// TIA Portal V17 export
// export: Created 2023-12-22T15:05:25.6828662Z, ExportSetting WithDefaults, DisplayName Totally Integrated Automation Portal, DisplayVersion V17, DisplayName TIA Portal Openness, DisplayVersion V17, DisplayName TIA Portal Version Control Interface, DisplayVersion V17, DisplayName STEP 7 Professional, DisplayVersion V17, DisplayName STEP 7 Safety, DisplayVersion V17, DisplayName WinCC Advanced, DisplayVersion V17
FUNCTION_BLOCK "Block_Line"   // FB12, LAD
{ S7_Optimized_Access := 'TRUE' }
VERSION : 0.1
// stored: AutoNumber true, IsIECCheckEnabled false, IsRetainMemResEnabled false, MemoryReserve 100, SetENOAutomatically false, UDAEnableTagReadback false
   VAR_INPUT
      Flow : Real;   // Расходомер принимающей трубы
      SP_C : Real := 0.01;   // Уставка дозации, % масс, 0.05-1
      PE : Real;   // Датчик давления
      ALLS : Bool;   // Авариййный нижний уровень бака
      RT : Bool;   // Ротаметр
      RM : Bool;   // Датчик протока вместо расходомера
      KC_ON : Bool;   // Клапан открыт
      PE_LLS : Bool;
      PE_HHS : Bool;
   END_VAR
   VAR_OUTPUT
      KC_CMD : Bool;   // Открытие клапана
   END_VAR
   VAR_IN_OUT
      Report_H : "Line_Report";   // Разовый отчёт
   END_VAR
   VAR RETAIN
      LINE_NUMBER : Int;   // номер линии
   END_VAR
   VAR
      Start : Bool;   // Запуск линии
      Main_ON : Bool;   // Команда основного насоса
      Reserv_ON : Bool;   // Команда резервного насоса
   END_VAR
   VAR RETAIN
      Hand { S7_SetPoint := 'True'} : Bool;   // 1 - Задание скорости насосов в ручном режиме
      Choice_Tank : Bool;   // 0 - основной танк, 1 - резервный
      SP_Source { S7_SetPoint := 'True'} : Bool;   // 0 - по формуле расчета, 1 - равен входу Flow
      PID_Not_Use { S7_SetPoint := 'True'} : Bool;   // Использовать ПИД (0 - использовать, 1 - не использовать)
      Mode { S7_SetPoint := 'True'} : Bool;   // 0 - без разбаления, 1 - с разбавлением
      Mode_Local : Bool;   // Режим: 0 - местный, 1 - локальный
   END_VAR
   VAR
      Res_CMD : Bool;   // Команда ротации по наработке
      Res_ANY : Bool;   // Первый насос в резерве
      No_Water : Bool;   // Авария "Нет продукта" HMI
      Dry_Run : Bool;   // Авария "Нет протока, сухой ход" HMI
      Pump_Main_Alarm : Bool;   // Выходной сигнал аварии насоса 1
      Pump_Reserv_Alarm : Bool;   // Выходной сигнал аварии насоса 2
      Main_Line_Ok : Bool := true;   // Готовность основной линии
      Low_Stop : Bool;   // Остановка по низкому протоку
      RM_1_Alarm : Bool;   // Авария основного расходомера
      RM_2_Alarm : Bool;   // Авария дополнительного расходомера
   END_VAR
   VAR RETAIN
      RM_1_Report_DI { S7_SetPoint := 'True'} : Bool;   // Использовать импусльный сигнал для отчётов
      RM_2_Report_DI { S7_SetPoint := 'True'} : Bool;   // Использовать импусльный сигнал для отчётов
      RM_Weight { S7_SetPoint := 'True'} : Real := 1.0;   // Вес импульса
   END_VAR
   VAR
      Status_Main : Int;   // Статус основного насоса
      Status_Reserv : Int;   // Статус резервного насоса
      Events : Word;   // События линии
      SP_A : Real;   // Уставка авторежима
   END_VAR
   VAR RETAIN
      SP_M { S7_SetPoint := 'True'} : Real;   // Уставка ручного режима
      SP_min { S7_SetPoint := 'True'} : Real := 10.0;   // Минимальная скорость насоса
      SP_max { S7_SetPoint := 'True'} : Real := 1000.0;   // Максимальная скорость насоса
      PE_min { S7_SetPoint := 'True'} : Real := 0.15;   // Низкое давление в линии
      PE_max { S7_SetPoint := 'True'} : Real := 2.5;   // Высокое давление в линии
   END_VAR
   VAR
      Pump_SP : Real;   // Актуальная скорость насоса
   END_VAR
   VAR RETAIN
      D { S7_SetPoint := 'True'} : Real;   // Уставка дозы
      D_Num : Real;   // Количество замерок дозы
      D_Sum : Real;   // Общаяя сумма дозы
   END_VAR
   VAR
      C : Real;   // Рабочие данные о концентрации
   END_VAR
   VAR RETAIN
      C_Tank { S7_SetPoint := 'True'} : Real;   // Концентрация в резервном баке
   END_VAR
   VAR
      Flow_Line : Real;   // Расходомер, используемый в данный момент
      Flow_s { ExternalAccessible := 'False'; ExternalVisible := 'False'; ExternalWritable := 'False'} : Real;   // Переведенный в секунды
      Alarm_SP : Real;   // Аварийный коэфф соотношение уставки к реальной скорости насоса
   END_VAR
   VAR RETAIN
      Low_Flow { S7_SetPoint := 'True'} : Real;   // Низкий проток в основной линии
      Res_Main : Real;   // Наработка основного насоса
      Res_Reserv : Real;   // Наработка резревного насоса
      Res_SP { S7_SetPoint := 'True'} : Real;   // Уставка переключения по наработке
   END_VAR
   VAR
      Last_D : Real;   // Предъдущее значение дозы
      Last_SP : Real;   // Предъдущее значение расхода
   END_VAR
   VAR RETAIN
      Use : Struct   // Конфигурация
         RT { S7_SetPoint := 'True'} : Bool;   // Использование ротаметра
         RM { S7_SetPoint := 'True'} : Bool;   // Использование датчика протока вместо расходомера
         SP { S7_SetPoint := 'True'} : Bool := true;   // Использовать аналоговое регулирование
         Flow { S7_SetPoint := 'True'} : Bool := true;   // Использовать контрольный расходомер
         Res { S7_SetPoint := 'True'} : Bool;   // Использовать переключение по наработке
         DME { S7_SetPoint := 'True'} : Bool;   // Мембранные насосы
         PE { S7_SetPoint := 'True'} : Bool;
      END_STRUCT;
   END_VAR
   VAR
      Messages : Struct   // - Аварийные сообщения
         Low_Duct : Bool;   // Авария - низкий проток
         Low_Conc : Bool;   // Авария - низкая концентрация
         RT_ON : Bool;   // Авария - нет протока воды на ротаметре
         RT_OFF : Bool;   // Авария - поток воды не пропал на ротаметре
         RM_Error : Bool;   // Авария - неисправен расходомер
         PE_Low : Bool;   // Авария - низкое давление в линии
         PE_High : Bool;   // Авария - высокое давление в линии
         Alarm : Word;   // Слово аварий для панели
      END_STRUCT;
      Messages_Cancel : Struct   // - Отмена остановки
         Low_Duct : Bool;   // Авария - низкий проток
         Low_Conc : Bool;   // Авария - низкая концентрация
         RT_ON : Bool;   // Авария - нет протока воды на ротаметре
         RT_OFF : Bool;   // Авария - поток воды не пропал на ротаметре
         PE_Low : Bool;   // Авария - низкое давление в линии
         PE_High : Bool;   // Авария - высокое давление в линии
      END_STRUCT;
      Messages_Stop : Struct   // - Остановка по аварии
         Low_Duct : Bool;   // Авария - низкий проток
         Low_Conc : Bool;   // Авария - низкая концентрация
         RT_ON : Bool;   // Авария - нет протока воды на ротаметре
         RT_OFF : Bool;   // Авария - поток воды не пропал на ротаметре
         PE_Low : Bool;   // Авария - низкое давление в линии
         PE_High : Bool;   // Авария - высокое давление в линии
      END_STRUCT;
      Messages_Counter : Struct   // - Счётчик аварийных срабатываний
         Low_Duct : Int;   // Авария - низкий проток
         Low_Conc : Int;   // Авария - низкая концентрация
         RT_ON : Int;   // Авария - нет протока воды на ротаметре
         RT_OFF : Int;   // Авария - поток воды не пропал на ротаметре
         PE_Low : Int;   // Авария - низкое давление в линии
         PE_High : Int;   // Авария - высокое давление в линии
      END_STRUCT;
      Messages_Reset : Struct   // - Сброс счётчика
         Low_Duct : Bool;   // Авария - низкий проток
         Low_Conc : Bool;   // Авария - низкая концентрация
         RT_ON : Bool;   // Авария - нет протока воды на ротаметре
         RT_OFF : Bool;   // Авария - поток воды не пропал на ротаметре
         PE_Low : Bool;   // Авария - низкое давление в линии
         PE_High : Bool;   // Авария - высокое давление в линии
      END_STRUCT;
      Messages_REQ_Stop : Struct   // - Запрос остановки по аварии
         Low_Duct : Bool;   // Авария - низкий проток
         Low_Conc : Bool;   // Авария - низкая концентрация
         RT_ON : Bool;   // Авария - нет протока воды на ротаметре
         RT_OFF : Bool;   // Авария - поток воды не пропал на ротаметре
         PE_Low : Bool;   // Авария - низкое давление в линии
         PE_High : Bool;   // Авария - высокое давление в линии
      END_STRUCT;
      Timers_Stop : Array[0..5] of "Time_M";   // Таймеры останова
      Timers_Alm : Array[0..5] of "Time_M";   // Таймеры аварий
      T_Main_Alarm : "Time_M";   // Авария основного насоса по датчику протока
      T_Reserv_Alarm : "Time_M";   // Авария резервного насоса по датчику протока
      T_Main_Line_Ok : "Time_M";   // Таймер готовности основной линии
      T_No_Water : "Time_M";   // Нет продукта в баке
      T_Dry_Run : "Time_M";   // Нет протока в линии
      pos : Array[0..15] of Bool;   // Вспомогательные переменные
      PID { S7_SetPoint := 'True'} : "PID_ex";
      FlowMeter_1 { S7_SetPoint := 'True'} : "DRV_Flow_old";   // Расход 1
      FlowMeter_2 { S7_SetPoint := 'True'} : "DRV_Flow_old";   // Расход 2
   END_VAR
   VAR_TEMP
      ev : Bool;
      x : Real;
   END_VAR
   VAR CONSTANT
      "1s" : Real := 0.00028;
      "1m" : Real := 0.017;
   END_VAR
   // // Report_H.Res_1 : Резерв 1
   // // Report_H.Res_2 : Резерв 2
   VAR_TEMP   // added for the SCL form of the ladder/FBD networks
      _w1 : Bool;
      _w2 : Bool;
      _w3 : Bool;
      _w4 : Bool;
      _w5 : Bool;
      _w6 : Bool;
      _w7 : Bool;
      _w8 : Bool;
      _w9 : Bool;
      _w10 : Bool;
      _w11 : Bool;
      _w12 : Bool;
      _w13 : Bool;
      _w14 : Bool;
   END_VAR
BEGIN

REGION Network 1: Режим: 0 - местный, 1 - локальный
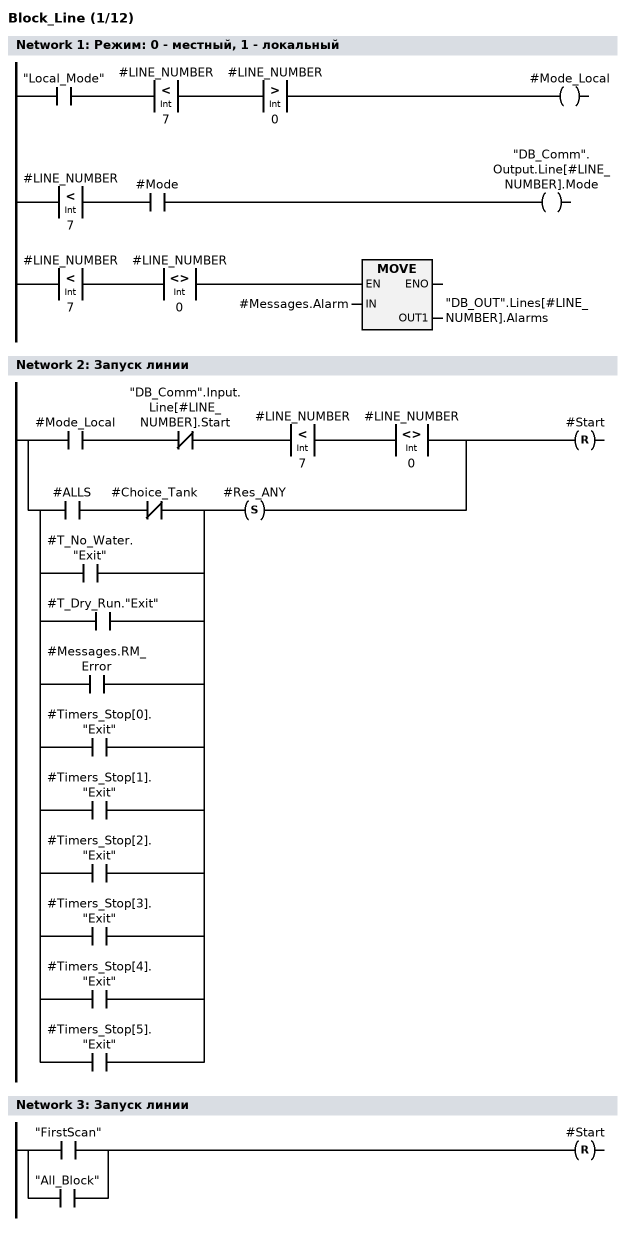
   RUNG wire#powerrail
      Contact( "Local_Mode" )
      { S7_Templates := "SrcType := Int" } LT_Contact(in1 := #LINE_NUMBER, in2 := 7)
      { S7_Templates := "SrcType := Int" } GT_Contact(in1 := #LINE_NUMBER, in2 := 0)
      Coil( #Mode_Local )
   END_RUNG
   RUNG wire#powerrail
      { S7_Templates := "SrcType := Int" } LT_Contact(in1 := #LINE_NUMBER, in2 := 7)
      Contact( #Mode )
      Coil( "DB_Comm".Output.Line[#LINE_NUMBER].Mode )
   END_RUNG
   RUNG wire#powerrail
      { S7_Templates := "SrcType := Int" } LT_Contact(in1 := #LINE_NUMBER, in2 := 7)
      { S7_Templates := "SrcType := Int" } NE_Contact(in1 := #LINE_NUMBER, in2 := 0)
      Move(in := #Messages.Alarm, out1 => "DB_OUT".Lines[#LINE_NUMBER].Alarms)
   END_RUNG
   // the same network as SCL:
   #Mode_Local := "Local_Mode" AND (#LINE_NUMBER < 7) AND (#LINE_NUMBER > 0);
   "DB_Comm".Output.Line[#LINE_NUMBER].Mode := (#LINE_NUMBER < 7) AND #Mode;
   IF (#LINE_NUMBER < 7) AND (#LINE_NUMBER <> 0) THEN
       "DB_OUT".Lines[#LINE_NUMBER].Alarms := #Messages.Alarm;
   END_IF;
END_REGION

REGION Network 2: Запуск линии
   RUNG wire#powerrail
      Contact( #Mode_Local )
      I_Contact( "DB_Comm".Input.Line[#LINE_NUMBER].Start )
      { S7_Templates := "SrcType := Int" } LT_Contact(in1 := #LINE_NUMBER, in2 := 7)
      { S7_Templates := "SrcType := Int" } NE_Contact(in1 := #LINE_NUMBER, in2 := 0)
      wire#w1
      R_Coil( #Start )
   END_RUNG
   RUNG wire#powerrail
      Contact( #ALLS )
      I_Contact( #Choice_Tank )
      wire#w2
      S_Coil( #Res_ANY )
   END_RUNG wire#w1
   RUNG wire#powerrail
      Contact( #T_No_Water."Exit" )
   END_RUNG wire#w2
   RUNG wire#powerrail
      Contact( #T_Dry_Run."Exit" )
   END_RUNG wire#w2
   RUNG wire#powerrail
      Contact( #Messages.RM_Error )
   END_RUNG wire#w2
   RUNG wire#powerrail
      Contact( #Timers_Stop[0]."Exit" )
   END_RUNG wire#w2
   RUNG wire#powerrail
      Contact( #Timers_Stop[1]."Exit" )
   END_RUNG wire#w2
   RUNG wire#powerrail
      Contact( #Timers_Stop[2]."Exit" )
   END_RUNG wire#w2
   RUNG wire#powerrail
      Contact( #Timers_Stop[3]."Exit" )
   END_RUNG wire#w2
   RUNG wire#powerrail
      Contact( #Timers_Stop[4]."Exit" )
   END_RUNG wire#w2
   RUNG wire#powerrail
      Contact( #Timers_Stop[5]."Exit" )
   END_RUNG wire#w2
   // the same network as SCL:
   #_w1 := (#ALLS AND NOT #Choice_Tank) OR #T_No_Water."Exit" OR #T_Dry_Run."Exit" OR #Messages.RM_Error OR #Timers_Stop[0]."Exit" OR #Timers_Stop[1]."Exit" OR #Timers_Stop[2]."Exit" OR #Timers_Stop[3]."Exit" OR #Timers_Stop[4]."Exit" OR #Timers_Stop[5]."Exit";
   IF #_w1 THEN #Res_ANY := TRUE; END_IF;
   IF (#Mode_Local AND NOT "DB_Comm".Input.Line[#LINE_NUMBER].Start AND (#LINE_NUMBER < 7) AND (#LINE_NUMBER <> 0)) OR #_w1 THEN
       #Start := FALSE;
   END_IF;
END_REGION

REGION Network 3: Запуск линии
   RUNG wire#powerrail
      Contact( "FirstScan" )
      wire#w1
      R_Coil( #Start )
   END_RUNG
   RUNG wire#powerrail
      Contact( "All_Block" )
   END_RUNG wire#w1
   // the same network as SCL:
   IF "FirstScan" OR "All_Block" THEN #Start := FALSE; END_IF;
END_REGION

REGION Network 4: Формирование событий линии
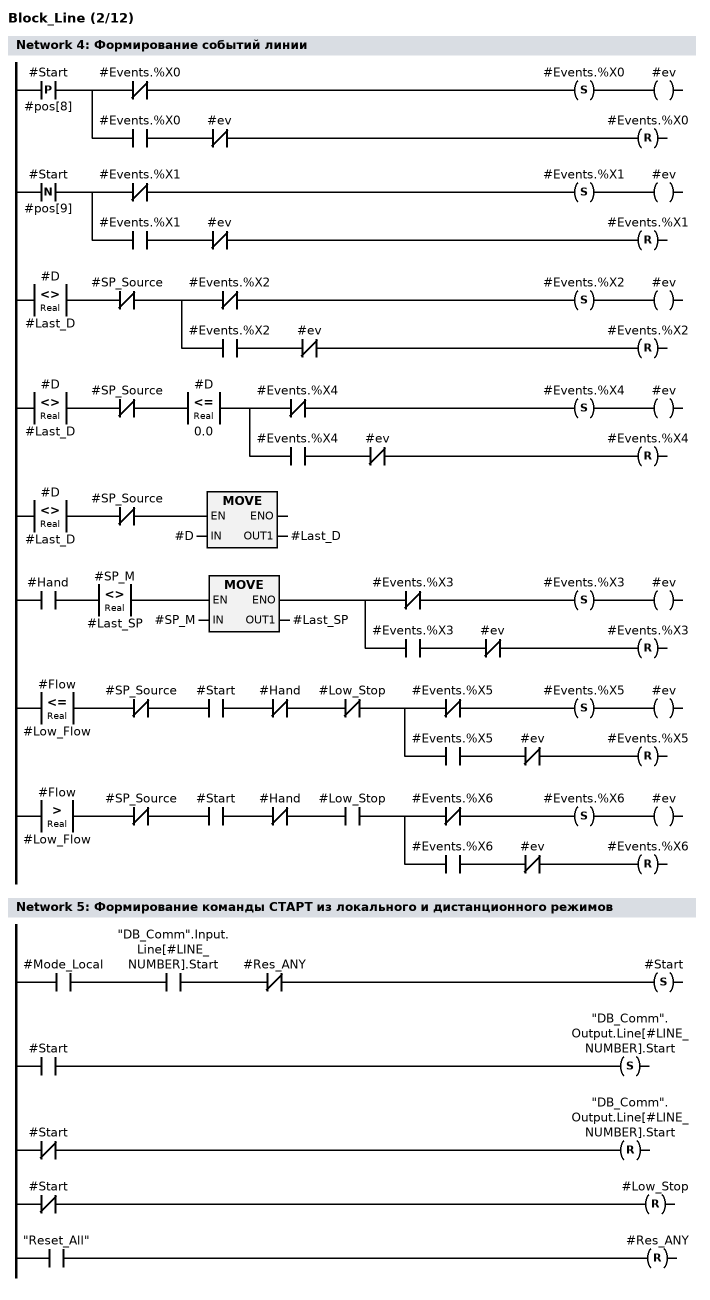
   RUNG wire#powerrail
      P_Contact(operand := #Start, bit := #pos[8])
      wire#w1
      I_Contact( #Events.%X0 )
      S_Coil( #Events.%X0 )
      Coil( #ev )
   END_RUNG
   RUNG wire#w1
      Contact( #Events.%X0 )
      I_Contact( #ev )
      R_Coil( #Events.%X0 )
   END_RUNG
   RUNG wire#powerrail
      N_Contact(operand := #Start, bit := #pos[9])
      wire#w2
      I_Contact( #Events.%X1 )
      S_Coil( #Events.%X1 )
      Coil( #ev )
   END_RUNG
   RUNG wire#w2
      Contact( #Events.%X1 )
      I_Contact( #ev )
      R_Coil( #Events.%X1 )
   END_RUNG
   RUNG wire#powerrail
      { S7_Templates := "SrcType := Real" } NE_Contact(in1 := #D, in2 := #Last_D)
      I_Contact( #SP_Source )
      wire#w3
      I_Contact( #Events.%X2 )
      S_Coil( #Events.%X2 )
      Coil( #ev )
   END_RUNG
   RUNG wire#w3
      Contact( #Events.%X2 )
      I_Contact( #ev )
      R_Coil( #Events.%X2 )
   END_RUNG
   RUNG wire#powerrail
      { S7_Templates := "SrcType := Real" } NE_Contact(in1 := #D, in2 := #Last_D)
      I_Contact( #SP_Source )
      { S7_Templates := "SrcType := Real" } LE_Contact(in1 := #D, in2 := 0.0)
      wire#w4
      I_Contact( #Events.%X4 )
      S_Coil( #Events.%X4 )
      Coil( #ev )
   END_RUNG
   RUNG wire#w4
      Contact( #Events.%X4 )
      I_Contact( #ev )
      R_Coil( #Events.%X4 )
   END_RUNG
   RUNG wire#powerrail
      { S7_Templates := "SrcType := Real" } NE_Contact(in1 := #D, in2 := #Last_D)
      I_Contact( #SP_Source )
      Move(in := #D, out1 => #Last_D)
   END_RUNG
   RUNG wire#powerrail
      Contact( #Hand )
      { S7_Templates := "SrcType := Real" } NE_Contact(in1 := #SP_M, in2 := #Last_SP)
      Move(in := #SP_M, out1 => #Last_SP)
      wire#w5
      I_Contact( #Events.%X3 )
      S_Coil( #Events.%X3 )
      Coil( #ev )
   END_RUNG
   RUNG wire#w5
      Contact( #Events.%X3 )
      I_Contact( #ev )
      R_Coil( #Events.%X3 )
   END_RUNG
   RUNG wire#powerrail
      { S7_Templates := "SrcType := Real" } LE_Contact(in1 := #Flow, in2 := #Low_Flow)
      I_Contact( #SP_Source )
      Contact( #Start )
      I_Contact( #Hand )
      I_Contact( #Low_Stop )
      wire#w6
      I_Contact( #Events.%X5 )
      S_Coil( #Events.%X5 )
      Coil( #ev )
   END_RUNG
   RUNG wire#w6
      Contact( #Events.%X5 )
      I_Contact( #ev )
      R_Coil( #Events.%X5 )
   END_RUNG
   RUNG wire#powerrail
      { S7_Templates := "SrcType := Real" } GT_Contact(in1 := #Flow, in2 := #Low_Flow)
      I_Contact( #SP_Source )
      Contact( #Start )
      I_Contact( #Hand )
      Contact( #Low_Stop )
      wire#w7
      I_Contact( #Events.%X6 )
      S_Coil( #Events.%X6 )
      Coil( #ev )
   END_RUNG
   RUNG wire#w7
      Contact( #Events.%X6 )
      I_Contact( #ev )
      R_Coil( #Events.%X6 )
   END_RUNG
   // the same network as SCL:
   #_w1 := #Start AND NOT #pos[8];   // rising edge of #Start
   #pos[8] := #Start;
   #_w2 := #_w1 AND NOT #Events.%X0;
   IF #_w2 THEN #Events.%X0 := TRUE; END_IF;
   #ev := #_w2;
   IF #_w1 AND #Events.%X0 AND NOT #ev THEN #Events.%X0 := FALSE; END_IF;
   #_w3 := NOT #Start AND #pos[9];   // falling edge of #Start
   #pos[9] := #Start;
   #_w4 := #_w3 AND NOT #Events.%X1;
   IF #_w4 THEN #Events.%X1 := TRUE; END_IF;
   #ev := #_w4;
   IF #_w3 AND #Events.%X1 AND NOT #ev THEN #Events.%X1 := FALSE; END_IF;
   #_w5 := (#D <> #Last_D) AND NOT #SP_Source;
   #_w6 := #_w5 AND NOT #Events.%X2;
   IF #_w6 THEN #Events.%X2 := TRUE; END_IF;
   #ev := #_w6;
   IF #_w5 AND #Events.%X2 AND NOT #ev THEN #Events.%X2 := FALSE; END_IF;
   #_w7 := (#D <> #Last_D) AND NOT #SP_Source AND (#D <= 0.0);
   #_w8 := #_w7 AND NOT #Events.%X4;
   IF #_w8 THEN #Events.%X4 := TRUE; END_IF;
   #ev := #_w8;
   IF #_w7 AND #Events.%X4 AND NOT #ev THEN #Events.%X4 := FALSE; END_IF;
   IF (#D <> #Last_D) AND NOT #SP_Source THEN #Last_D := #D; END_IF;
   #_w9 := #Hand AND (#SP_M <> #Last_SP);
   IF #_w9 THEN #Last_SP := #SP_M; END_IF;
   #_w10 := #_w9 AND NOT #Events.%X3;
   IF #_w10 THEN #Events.%X3 := TRUE; END_IF;
   #ev := #_w10;
   IF #_w9 AND #Events.%X3 AND NOT #ev THEN #Events.%X3 := FALSE; END_IF;
   #_w11 := (#Flow <= #Low_Flow) AND NOT #SP_Source AND #Start AND NOT #Hand AND NOT #Low_Stop;
   #_w12 := #_w11 AND NOT #Events.%X5;
   IF #_w12 THEN #Events.%X5 := TRUE; END_IF;
   #ev := #_w12;
   IF #_w11 AND #Events.%X5 AND NOT #ev THEN #Events.%X5 := FALSE; END_IF;
   #_w13 := (#Flow > #Low_Flow) AND NOT #SP_Source AND #Start AND NOT #Hand AND #Low_Stop;
   #_w14 := #_w13 AND NOT #Events.%X6;
   IF #_w14 THEN #Events.%X6 := TRUE; END_IF;
   #ev := #_w14;
   IF #_w13 AND #Events.%X6 AND NOT #ev THEN #Events.%X6 := FALSE; END_IF;
END_REGION

REGION Network 5: Формирование команды СТАРТ из локального и дистанционного режимов
   RUNG wire#powerrail
      Contact( #Mode_Local )
      Contact( "DB_Comm".Input.Line[#LINE_NUMBER].Start )
      I_Contact( #Res_ANY )
      S_Coil( #Start )
   END_RUNG
   RUNG wire#powerrail
      Contact( #Start )
      S_Coil( "DB_Comm".Output.Line[#LINE_NUMBER].Start )
   END_RUNG
   RUNG wire#powerrail
      I_Contact( #Start )
      R_Coil( "DB_Comm".Output.Line[#LINE_NUMBER].Start )
   END_RUNG
   RUNG wire#powerrail
      I_Contact( #Start )
      R_Coil( #Low_Stop )
   END_RUNG
   RUNG wire#powerrail
      Contact( "Reset_All" )
      R_Coil( #Res_ANY )
   END_RUNG
   // the same network as SCL:
   IF #Mode_Local AND "DB_Comm".Input.Line[#LINE_NUMBER].Start AND NOT #Res_ANY THEN #Start := TRUE; END_IF;
   IF #Start THEN "DB_Comm".Output.Line[#LINE_NUMBER].Start := TRUE; END_IF;
   IF NOT #Start THEN
       "DB_Comm".Output.Line[#LINE_NUMBER].Start := FALSE;
       #Low_Stop := FALSE;
   END_IF;
   IF "Reset_All" THEN #Res_ANY := FALSE; END_IF;
END_REGION

REGION Network 6: Старт - выбора насоса
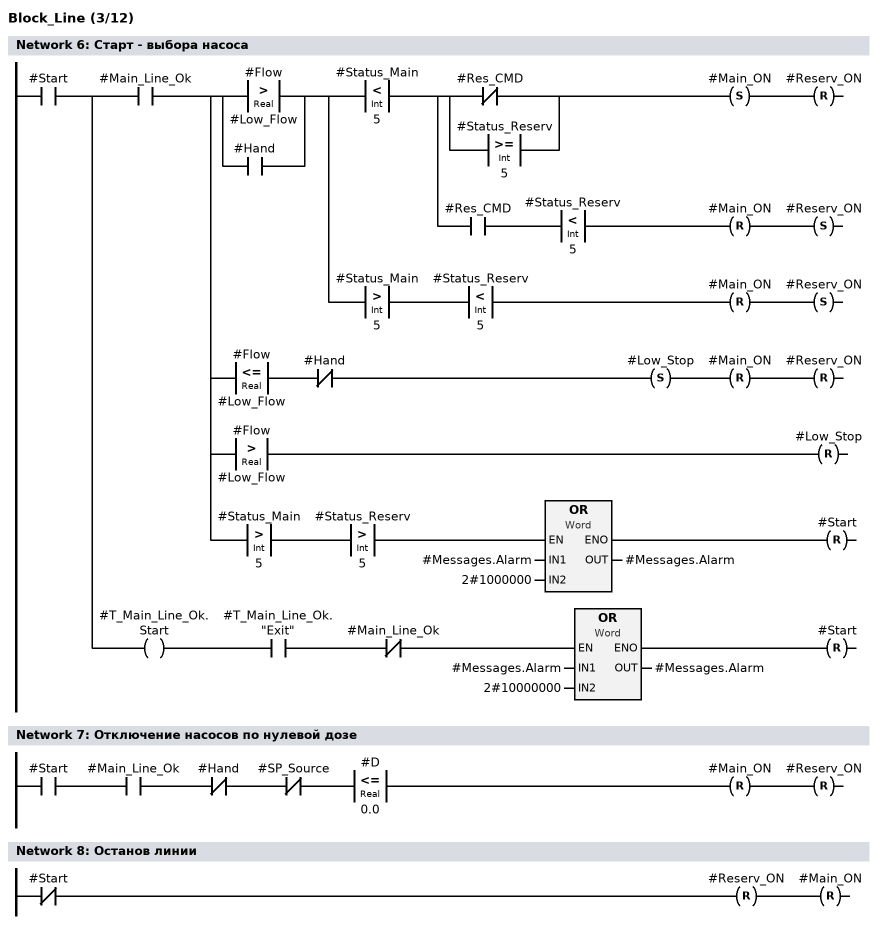
   #_w1 := #Start AND #Main_Line_Ok;
   #_w2 := #_w1 AND ((#Flow > #Low_Flow) OR #Hand);
   #_w3 := #_w2 AND (#Status_Main < 5);
   IF #_w3 AND (NOT #Res_CMD OR (#Status_Reserv >= 5)) THEN
       #Main_ON := TRUE;
       #Reserv_ON := FALSE;
   END_IF;
   IF #_w3 AND #Res_CMD AND (#Status_Reserv < 5) THEN
       #Main_ON := FALSE;
       #Reserv_ON := TRUE;
   END_IF;
   IF #_w2 AND (#Status_Main > 5) AND (#Status_Reserv < 5) THEN
       #Main_ON := FALSE;
       #Reserv_ON := TRUE;
   END_IF;
   IF #_w1 AND (#Flow <= #Low_Flow) AND NOT #Hand THEN
       #Low_Stop := TRUE;
       #Main_ON := FALSE;
       #Reserv_ON := FALSE;
   END_IF;
   IF #_w1 AND (#Flow > #Low_Flow) THEN #Low_Stop := FALSE; END_IF;
   IF #_w1 AND (#Status_Main > 5) AND (#Status_Reserv > 5) THEN
       #Messages.Alarm := #Messages.Alarm OR 2#1000000;
   END_IF;
   #_w4 := #Start;
   IF #_w1 AND (#Status_Main > 5) AND (#Status_Reserv > 5) THEN #Start := FALSE; END_IF;
   #T_Main_Line_Ok.Start := #_w4;
   IF #_w4 AND #T_Main_Line_Ok."Exit" AND NOT #Main_Line_Ok THEN
       #Messages.Alarm := #Messages.Alarm OR 2#10000000;
       #Start := FALSE;
   END_IF;
END_REGION

REGION Network 7: Отключение насосов по нулевой дозе
   RUNG wire#powerrail
      Contact( #Start )
      Contact( #Main_Line_Ok )
      I_Contact( #Hand )
      I_Contact( #SP_Source )
      { S7_Templates := "SrcType := Real" } LE_Contact(in1 := #D, in2 := 0.0)
      R_Coil( #Main_ON )
      R_Coil( #Reserv_ON )
   END_RUNG
   // the same network as SCL:
   IF #Start AND #Main_Line_Ok AND NOT #Hand AND NOT #SP_Source AND (#D <= 0.0) THEN
       #Main_ON := FALSE;
       #Reserv_ON := FALSE;
   END_IF;
END_REGION

REGION Network 8: Останов линии
   RUNG wire#powerrail
      I_Contact( #Start )
      R_Coil( #Reserv_ON )
      R_Coil( #Main_ON )
   END_RUNG
   // the same network as SCL:
   IF NOT #Start THEN
       #Reserv_ON := FALSE;
       #Main_ON := FALSE;
   END_IF;
END_REGION

REGION Network 9: Подсчёт наработки насосов и управление выбором основного и резервного
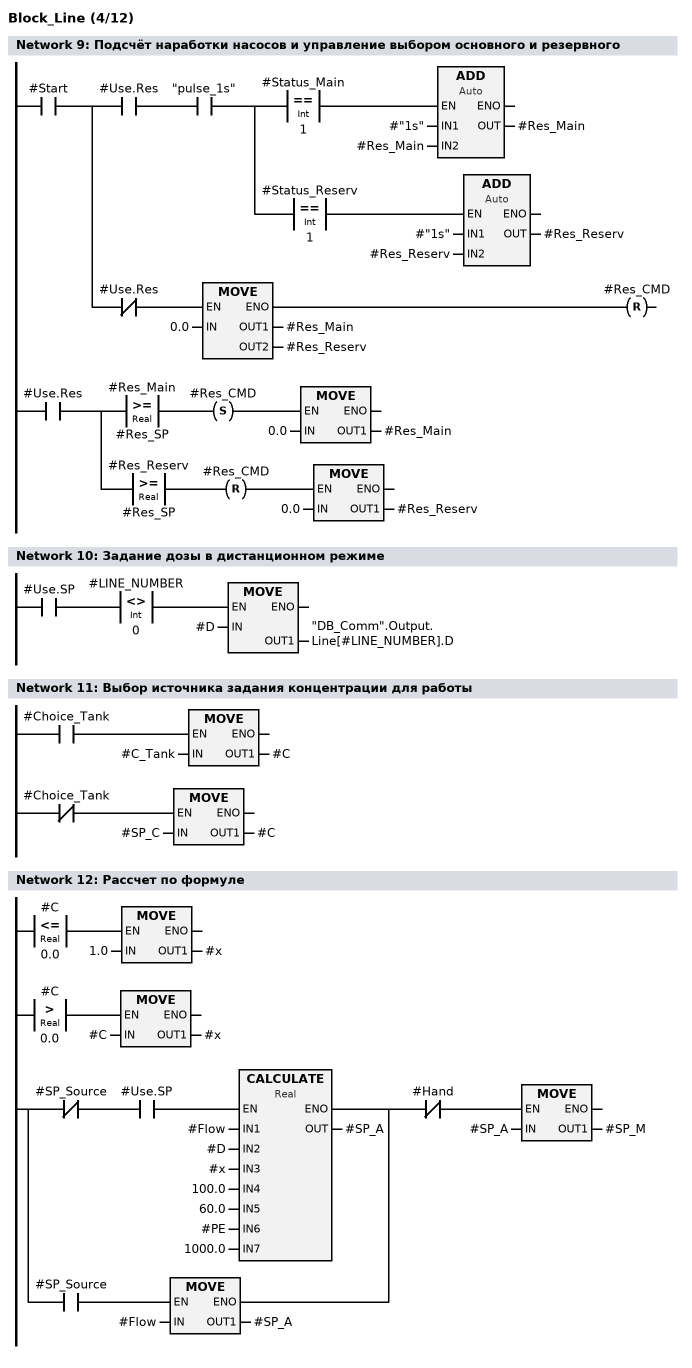
   RUNG wire#powerrail
      Contact( #Start )
      wire#w1
      Contact( #Use.Res )
      Contact( "pulse_1s" )
      wire#w2
      { S7_Templates := "SrcType := Int" } EQ_Contact(in1 := #Status_Main, in2 := 1)
      Add(in1 := #"1s", in2 := #Res_Main, out => #Res_Main)
   END_RUNG
   RUNG wire#w2
      { S7_Templates := "SrcType := Int" } EQ_Contact(in1 := #Status_Reserv, in2 := 1)
      Add(in1 := #"1s", in2 := #Res_Reserv, out => #Res_Reserv)
   END_RUNG
   RUNG wire#w1
      I_Contact( #Use.Res )
      Move(in := 0.0, out1 => #Res_Main, out2 => #Res_Reserv)
      R_Coil( #Res_CMD )
   END_RUNG
   RUNG wire#powerrail
      Contact( #Use.Res )
      wire#w3
      { S7_Templates := "SrcType := Real" } GE_Contact(in1 := #Res_Main, in2 := #Res_SP)
      S_Coil( #Res_CMD )
      Move(in := 0.0, out1 => #Res_Main)
   END_RUNG
   RUNG wire#w3
      { S7_Templates := "SrcType := Real" } GE_Contact(in1 := #Res_Reserv, in2 := #Res_SP)
      R_Coil( #Res_CMD )
      Move(in := 0.0, out1 => #Res_Reserv)
   END_RUNG
   // the same network as SCL:
   #_w1 := #Start AND #Use.Res AND "pulse_1s";
   IF #_w1 AND (#Status_Main = 1) THEN #Res_Main := #"1s" + #Res_Main; END_IF;
   IF #_w1 AND (#Status_Reserv = 1) THEN #Res_Reserv := #"1s" + #Res_Reserv; END_IF;
   IF #Start AND NOT #Use.Res THEN
       #Res_Main := 0.0;
       #Res_Reserv := 0.0;
       #Res_CMD := FALSE;
   END_IF;
   IF #Use.Res AND (#Res_Main >= #Res_SP) THEN
       #Res_CMD := TRUE;
       #Res_Main := 0.0;
   END_IF;
   IF #Use.Res AND (#Res_Reserv >= #Res_SP) THEN
       #Res_CMD := FALSE;
       #Res_Reserv := 0.0;
   END_IF;
END_REGION

REGION Network 10: Задание дозы в дистанционном режиме
   RUNG wire#powerrail
      Contact( #Use.SP )
      { S7_Templates := "SrcType := Int" } NE_Contact(in1 := #LINE_NUMBER, in2 := 0)
      Move(in := #D, out1 => "DB_Comm".Output.Line[#LINE_NUMBER].D)
   END_RUNG
   // the same network as SCL:
   IF #Use.SP AND (#LINE_NUMBER <> 0) THEN "DB_Comm".Output.Line[#LINE_NUMBER].D := #D; END_IF;
END_REGION

REGION Network 11: Выбор источника задания концентрации для работы
   RUNG wire#powerrail
      Contact( #Choice_Tank )
      Move(in := #C_Tank, out1 => #C)
   END_RUNG
   RUNG wire#powerrail
      I_Contact( #Choice_Tank )
      Move(in := #SP_C, out1 => #C)
   END_RUNG
   // the same network as SCL:
   IF #Choice_Tank THEN #C := #C_Tank; END_IF;
   IF NOT #Choice_Tank THEN #C := #SP_C; END_IF;
END_REGION

REGION Network 12: Рассчет по формуле
   RUNG wire#powerrail
      { S7_Templates := "SrcType := Real" } LE_Contact(in1 := #C, in2 := 0.0)
      Move(in := 1.0, out1 => #x)
   END_RUNG
   RUNG wire#powerrail
      { S7_Templates := "SrcType := Real" } GT_Contact(in1 := #C, in2 := 0.0)
      Move(in := #C, out1 => #x)
   END_RUNG
   RUNG wire#powerrail
      I_Contact( #SP_Source )
      Contact( #Use.SP )
      { S7_Templates := "SrcType := Real"; S7_Expression := "(IN2 * IN1) / ( IN3 / IN4) / (IN6 * IN7) / IN5" } Calculate(in1 := #Flow, in2 := #D, in3 := #x, in4 := 100.0, in5 := 60.0, in6 := #PE, in7 := 1000.0, out => #SP_A)
      wire#w1
      I_Contact( #Hand )
      Move(in := #SP_A, out1 => #SP_M)
   END_RUNG
   RUNG wire#powerrail
      Contact( #SP_Source )
      Move(in := #Flow, out1 => #SP_A)
   END_RUNG wire#w1
   // the same network as SCL:
   IF #C <= 0.0 THEN #x := 1.0; END_IF;
   IF #C > 0.0 THEN #x := #C; END_IF;
   #_w1 := NOT #SP_Source AND #Use.SP;
   IF #_w1 THEN #SP_A := (#D * #Flow) / ( #x / 100.0) / (#PE * 1000.0) / 60.0; END_IF;
   IF #SP_Source THEN #SP_A := #Flow; END_IF;
   IF (#_w1 OR #SP_Source) AND NOT #Hand THEN #SP_M := #SP_A; END_IF;
END_REGION

REGION Network 13: Выбор режима с разбавлением или без разбавления в дистанционном режиме
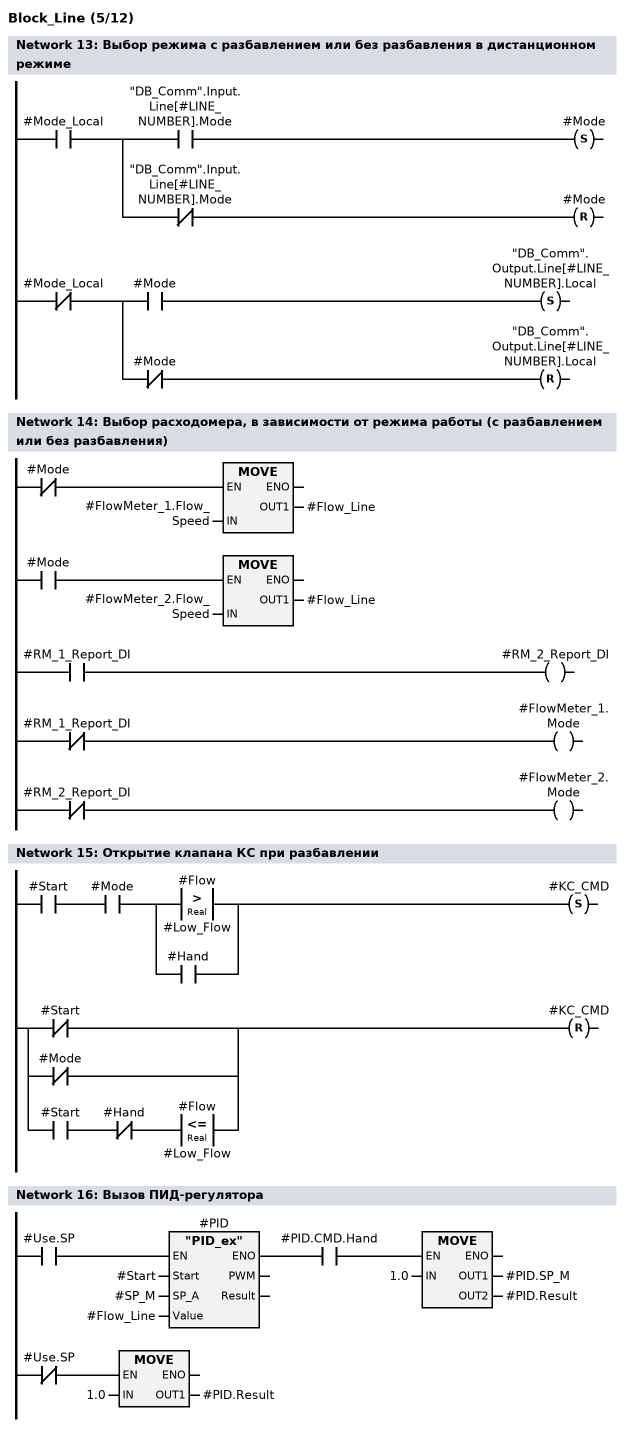
   RUNG wire#powerrail
      Contact( #Mode_Local )
      wire#w1
      Contact( "DB_Comm".Input.Line[#LINE_NUMBER].Mode )
      S_Coil( #Mode )
   END_RUNG
   RUNG wire#w1
      I_Contact( "DB_Comm".Input.Line[#LINE_NUMBER].Mode )
      R_Coil( #Mode )
   END_RUNG
   RUNG wire#powerrail
      I_Contact( #Mode_Local )
      wire#w2
      Contact( #Mode )
      S_Coil( "DB_Comm".Output.Line[#LINE_NUMBER].Local )
   END_RUNG
   RUNG wire#w2
      I_Contact( #Mode )
      R_Coil( "DB_Comm".Output.Line[#LINE_NUMBER].Local )
   END_RUNG
   // the same network as SCL:
   IF #Mode_Local AND "DB_Comm".Input.Line[#LINE_NUMBER].Mode THEN #Mode := TRUE; END_IF;
   IF #Mode_Local AND NOT "DB_Comm".Input.Line[#LINE_NUMBER].Mode THEN #Mode := FALSE; END_IF;
   IF NOT #Mode_Local AND #Mode THEN "DB_Comm".Output.Line[#LINE_NUMBER].Local := TRUE; END_IF;
   IF NOT #Mode_Local AND NOT #Mode THEN "DB_Comm".Output.Line[#LINE_NUMBER].Local := FALSE; END_IF;
END_REGION

REGION Network 14: Выбор расходомера, в зависимости от режима работы (с разбавлением или без разбавления)
   RUNG wire#powerrail
      I_Contact( #Mode )
      Move(in := #FlowMeter_1.Flow_Speed, out1 => #Flow_Line)
   END_RUNG
   RUNG wire#powerrail
      Contact( #Mode )
      Move(in := #FlowMeter_2.Flow_Speed, out1 => #Flow_Line)
   END_RUNG
   RUNG wire#powerrail
      Contact( #RM_1_Report_DI )
      Coil( #RM_2_Report_DI )
   END_RUNG
   RUNG wire#powerrail
      I_Contact( #RM_1_Report_DI )
      Coil( #FlowMeter_1.Mode )
   END_RUNG
   RUNG wire#powerrail
      I_Contact( #RM_2_Report_DI )
      Coil( #FlowMeter_2.Mode )
   END_RUNG
   // the same network as SCL:
   IF NOT #Mode THEN #Flow_Line := #FlowMeter_1.Flow_Speed; END_IF;
   IF #Mode THEN #Flow_Line := #FlowMeter_2.Flow_Speed; END_IF;
   #RM_2_Report_DI := #RM_1_Report_DI;
   #FlowMeter_1.Mode := NOT #RM_1_Report_DI;
   #FlowMeter_2.Mode := NOT #RM_2_Report_DI;
END_REGION

REGION Network 15: Открытие клапана КС при разбавлении
   RUNG wire#powerrail
      Contact( #Start )
      Contact( #Mode )
      wire#w1
      { S7_Templates := "SrcType := Real" } GT_Contact(in1 := #Flow, in2 := #Low_Flow)
      wire#w2
      S_Coil( #KC_CMD )
   END_RUNG
   RUNG wire#w1
      Contact( #Hand )
   END_RUNG wire#w2
   RUNG wire#powerrail
      I_Contact( #Start )
      wire#w3
      R_Coil( #KC_CMD )
   END_RUNG
   RUNG wire#powerrail
      I_Contact( #Mode )
   END_RUNG wire#w3
   RUNG wire#powerrail
      Contact( #Start )
      I_Contact( #Hand )
      { S7_Templates := "SrcType := Real" } LE_Contact(in1 := #Flow, in2 := #Low_Flow)
   END_RUNG wire#w3
   // the same network as SCL:
   IF #Start AND #Mode AND ((#Flow > #Low_Flow) OR #Hand) THEN #KC_CMD := TRUE; END_IF;
   IF NOT #Start OR NOT #Mode OR (#Start AND NOT #Hand AND (#Flow <= #Low_Flow)) THEN
       #KC_CMD := FALSE;
   END_IF;
END_REGION

REGION Network 16: Вызов ПИД-регулятора
   RUNG wire#powerrail
      Contact( #Use.SP )
      #PID(Start := #Start, SP_A := #SP_M, Value := #Flow_Line, PWM =>, Result =>)
      Contact( #PID.CMD.Hand )
      Move(in := 1.0, out1 => #PID.SP_M, out2 => #PID.Result)
   END_RUNG
   RUNG wire#powerrail
      I_Contact( #Use.SP )
      Move(in := 1.0, out1 => #PID.Result)
   END_RUNG
   // the same network as SCL:
   #PID(EN := #Use.SP, Start := #Start, SP_A := #SP_M, Value := #Flow_Line, ENO => #_w1);   // "PID_ex"
   IF #_w1 AND #PID.CMD.Hand THEN
       #PID.SP_M := 1.0;
       #PID.Result := 1.0;
   END_IF;
   IF NOT #Use.SP THEN #PID.Result := 1.0; END_IF;
END_REGION

REGION Network 17: Обнуление уставки при отстутствии аналогового управления насосами
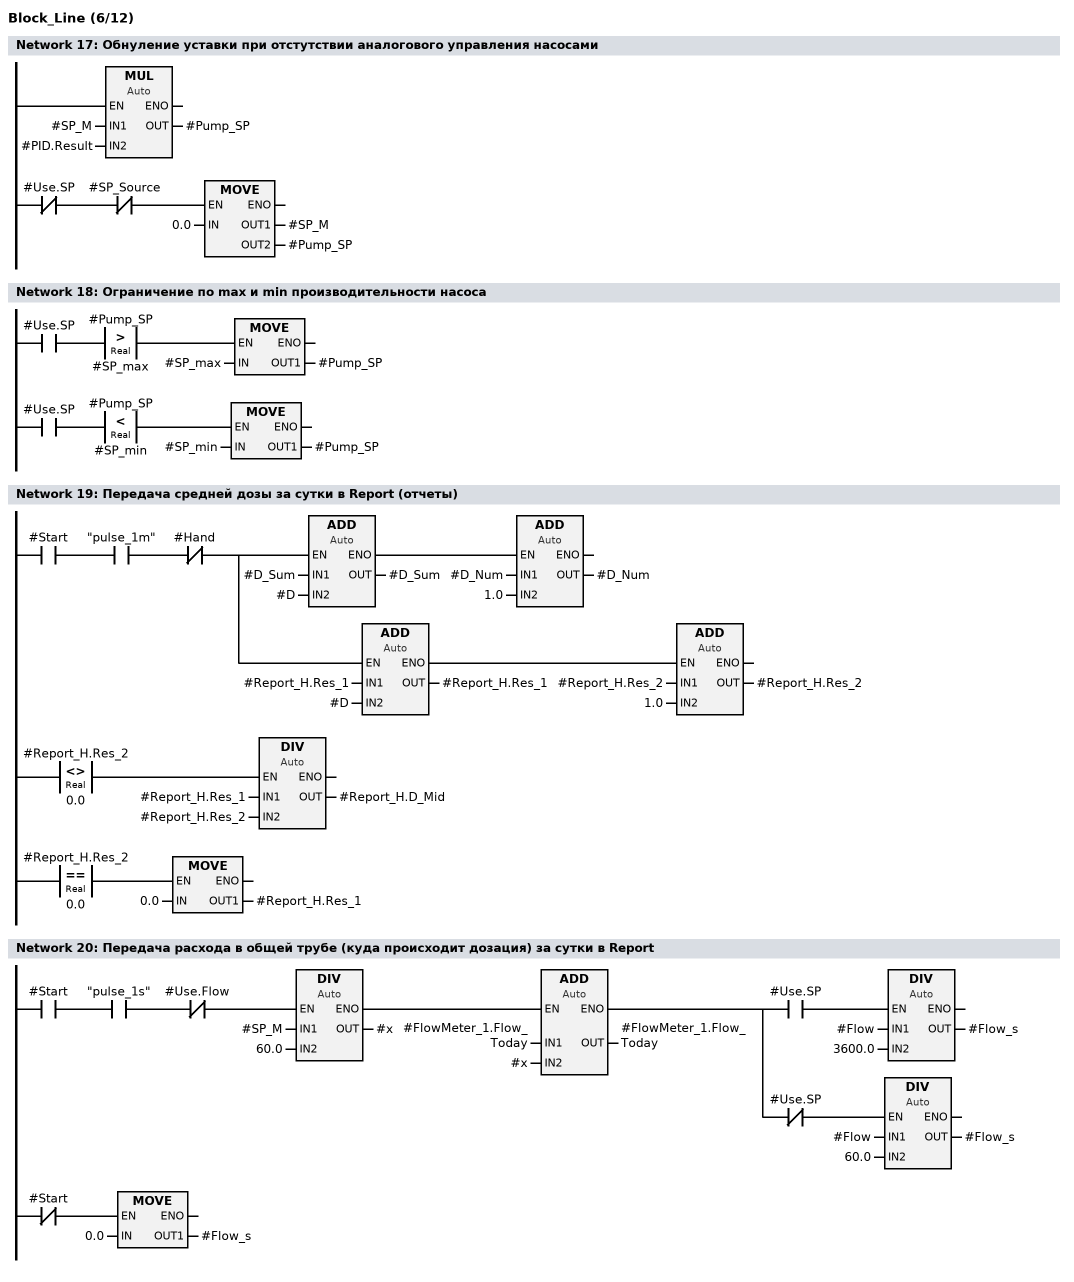
   RUNG wire#powerrail
      Mul(in1 := #SP_M, in2 := #PID.Result, out => #Pump_SP)
   END_RUNG
   RUNG wire#powerrail
      I_Contact( #Use.SP )
      I_Contact( #SP_Source )
      Move(in := 0.0, out1 => #SP_M, out2 => #Pump_SP)
   END_RUNG
   // the same network as SCL:
   #Pump_SP := #SP_M * #PID.Result;
   IF NOT #Use.SP AND NOT #SP_Source THEN
       #SP_M := 0.0;
       #Pump_SP := 0.0;
   END_IF;
END_REGION

REGION Network 18: Ограничение по max и min производительности насоса
   RUNG wire#powerrail
      Contact( #Use.SP )
      { S7_Templates := "SrcType := Real" } GT_Contact(in1 := #Pump_SP, in2 := #SP_max)
      Move(in := #SP_max, out1 => #Pump_SP)
   END_RUNG
   RUNG wire#powerrail
      Contact( #Use.SP )
      { S7_Templates := "SrcType := Real" } LT_Contact(in1 := #Pump_SP, in2 := #SP_min)
      Move(in := #SP_min, out1 => #Pump_SP)
   END_RUNG
   // the same network as SCL:
   IF #Use.SP AND (#Pump_SP > #SP_max) THEN #Pump_SP := #SP_max; END_IF;
   IF #Use.SP AND (#Pump_SP < #SP_min) THEN #Pump_SP := #SP_min; END_IF;
END_REGION

REGION Network 19: Передача средней дозы за сутки в Report (отчеты)
   RUNG wire#powerrail
      Contact( #Start )
      Contact( "pulse_1m" )
      I_Contact( #Hand )
      wire#w1
      Add(in1 := #D_Sum, in2 := #D, out => #D_Sum)
      Add(in1 := #D_Num, in2 := 1.0, out => #D_Num)
   END_RUNG
   RUNG wire#w1
      Add(in1 := #Report_H.Res_1, in2 := #D, out => #Report_H.Res_1)
      Add(in1 := #Report_H.Res_2, in2 := 1.0, out => #Report_H.Res_2)
   END_RUNG
   RUNG wire#powerrail
      { S7_Templates := "SrcType := Real" } NE_Contact(in1 := #Report_H.Res_2, in2 := 0.0)
      Div(in1 := #Report_H.Res_1, in2 := #Report_H.Res_2, out => #Report_H.D_Mid)
   END_RUNG
   RUNG wire#powerrail
      { S7_Templates := "SrcType := Real" } EQ_Contact(in1 := #Report_H.Res_2, in2 := 0.0)
      Move(in := 0.0, out1 => #Report_H.Res_1)
   END_RUNG
   // the same network as SCL:
   IF #Start AND "pulse_1m" AND NOT #Hand THEN
       #D_Sum := #D_Sum + #D;
       #D_Num := #D_Num + 1.0;
       #Report_H.Res_1 := #Report_H.Res_1 + #D;
       #Report_H.Res_2 := #Report_H.Res_2 + 1.0;
   END_IF;
   IF #Report_H.Res_2 <> 0.0 THEN #Report_H.D_Mid := #Report_H.Res_1 / #Report_H.Res_2; END_IF;
   IF #Report_H.Res_2 = 0.0 THEN #Report_H.Res_1 := 0.0; END_IF;
END_REGION

REGION Network 20: Передача расхода в общей трубе (куда происходит дозация) за сутки в Report
   RUNG wire#powerrail
      Contact( #Start )
      Contact( "pulse_1s" )
      I_Contact( #Use.Flow )
      Div(in1 := #SP_M, in2 := 60.0, out => #x)
      Add(in1 := #FlowMeter_1.Flow_Today, in2 := #x, out => #FlowMeter_1.Flow_Today)
      wire#w1
      Contact( #Use.SP )
      Div(in1 := #Flow, in2 := 3600.0, out => #Flow_s)
   END_RUNG
   RUNG wire#w1
      I_Contact( #Use.SP )
      Div(in1 := #Flow, in2 := 60.0, out => #Flow_s)
   END_RUNG
   RUNG wire#powerrail
      I_Contact( #Start )
      Move(in := 0.0, out1 => #Flow_s)
   END_RUNG
   // the same network as SCL:
   #_w1 := #Start AND "pulse_1s" AND NOT #Use.Flow;
   IF #_w1 THEN
       #x := #SP_M / 60.0;
       #FlowMeter_1.Flow_Today := #FlowMeter_1.Flow_Today + #x;
   END_IF;
   IF #_w1 AND #Use.SP THEN #Flow_s := #Flow / 3600.0; END_IF;
   IF #_w1 AND NOT #Use.SP THEN #Flow_s := #Flow / 60.0; END_IF;
   IF NOT #Start THEN #Flow_s := 0.0; END_IF;
END_REGION

REGION Network 21: Авария основного насоса по датчику протока
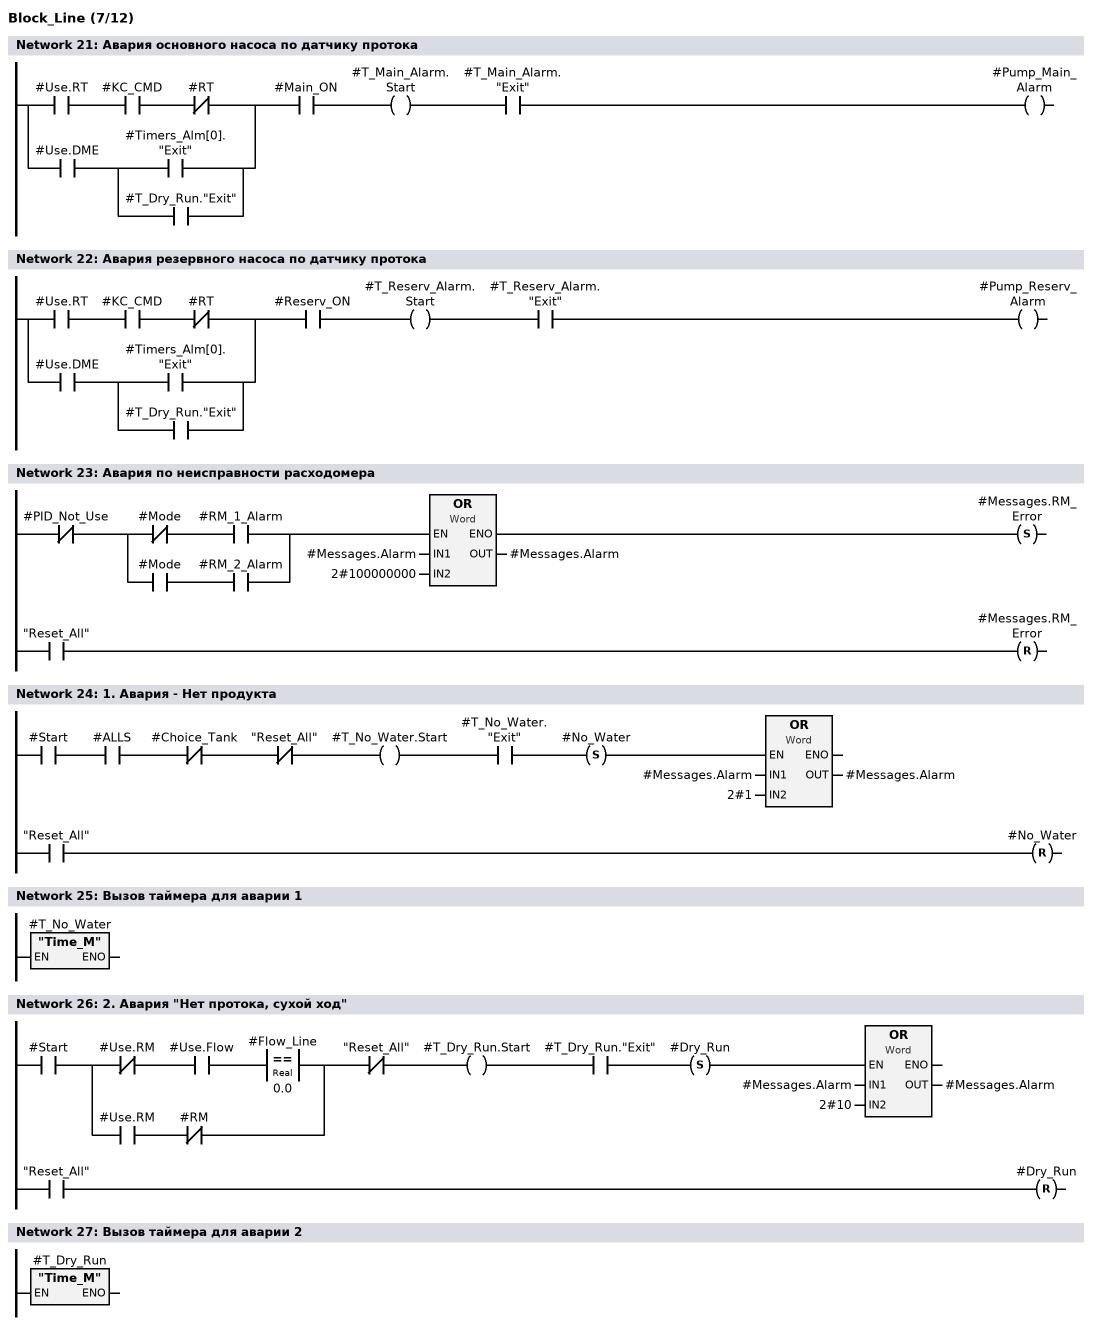
   RUNG wire#powerrail
      Contact( #Use.RT )
      Contact( #KC_CMD )
      I_Contact( #RT )
      wire#w1
      Contact( #Main_ON )
      Coil( #T_Main_Alarm.Start )
      Contact( #T_Main_Alarm."Exit" )
      Coil( #Pump_Main_Alarm )
   END_RUNG
   RUNG wire#powerrail
      Contact( #Use.DME )
      wire#w2
      Contact( #Timers_Alm[0]."Exit" )
   END_RUNG wire#w1
   RUNG wire#w2
      Contact( #T_Dry_Run."Exit" )
   END_RUNG wire#w1
   // the same network as SCL:
   #T_Main_Alarm.Start := ((#Use.RT AND #KC_CMD AND NOT #RT) OR (#Use.DME AND (#Timers_Alm[0]."Exit" OR #T_Dry_Run."Exit"))) AND #Main_ON;
   #Pump_Main_Alarm := #T_Main_Alarm.Start AND #T_Main_Alarm."Exit";
END_REGION

REGION Network 22: Авария резервного насоса по датчику протока
   RUNG wire#powerrail
      Contact( #Use.RT )
      Contact( #KC_CMD )
      I_Contact( #RT )
      wire#w1
      Contact( #Reserv_ON )
      Coil( #T_Reserv_Alarm.Start )
      Contact( #T_Reserv_Alarm."Exit" )
      Coil( #Pump_Reserv_Alarm )
   END_RUNG
   RUNG wire#powerrail
      Contact( #Use.DME )
      wire#w2
      Contact( #Timers_Alm[0]."Exit" )
   END_RUNG wire#w1
   RUNG wire#w2
      Contact( #T_Dry_Run."Exit" )
   END_RUNG wire#w1
   // the same network as SCL:
   #T_Reserv_Alarm.Start := ((#Use.RT AND #KC_CMD AND NOT #RT) OR (#Use.DME AND (#Timers_Alm[0]."Exit" OR #T_Dry_Run."Exit"))) AND #Reserv_ON;
   #Pump_Reserv_Alarm := #T_Reserv_Alarm.Start AND #T_Reserv_Alarm."Exit";
END_REGION

REGION Network 23: Авария по неисправности расходомера
   IF NOT #PID_Not_Use AND ((NOT #Mode AND #RM_1_Alarm) OR (#Mode AND #RM_2_Alarm)) THEN
       #Messages.Alarm := #Messages.Alarm OR 2#100000000;
       #Messages.RM_Error := TRUE;
   END_IF;
   IF "Reset_All" THEN #Messages.RM_Error := FALSE; END_IF;
END_REGION

REGION Network 24: 1. Авария - Нет продукта
   #T_No_Water.Start := #Start AND #ALLS AND NOT #Choice_Tank AND NOT "Reset_All";
   IF #T_No_Water.Start AND #T_No_Water."Exit" THEN
       #No_Water := TRUE;
       #Messages.Alarm := #Messages.Alarm OR 2#1;
   END_IF;
   IF "Reset_All" THEN #No_Water := FALSE; END_IF;
END_REGION

REGION Network 25: Вызов таймера для аварии 1
   RUNG wire#powerrail
      #T_No_Water()
   END_RUNG
   // the same network as SCL:
   #T_No_Water();   // "Time_M"
END_REGION

REGION Network 26: 2. Авария "Нет протока, сухой ход"
   #T_Dry_Run.Start := #Start AND ((NOT #Use.RM AND #Use.Flow AND (#Flow_Line = 0.0)) OR (#Use.RM AND NOT #RM)) AND NOT "Reset_All";
   IF #T_Dry_Run.Start AND #T_Dry_Run."Exit" THEN
       #Dry_Run := TRUE;
       #Messages.Alarm := #Messages.Alarm OR 2#10;
   END_IF;
   IF "Reset_All" THEN #Dry_Run := FALSE; END_IF;
END_REGION

REGION Network 27: Вызов таймера для аварии 2
   RUNG wire#powerrail
      #T_Dry_Run()
   END_RUNG
   // the same network as SCL:
   #T_Dry_Run();   // "Time_M"
END_REGION

REGION Network 28: 3. Авария - низкий проток
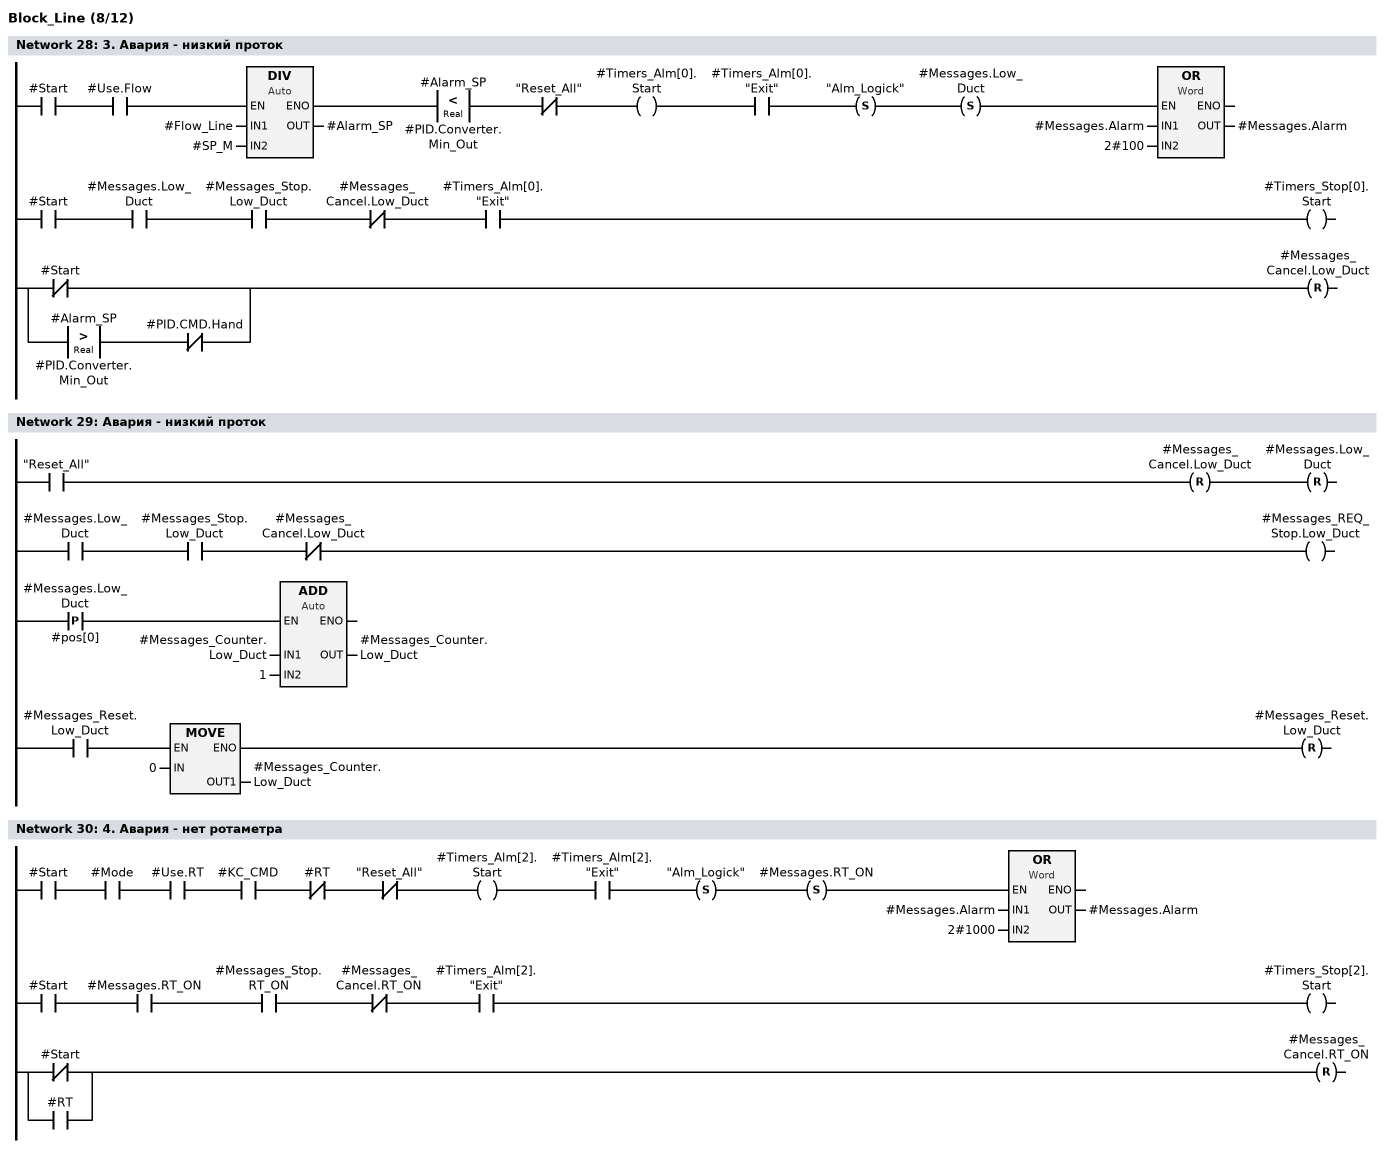
   #_w1 := #Start AND #Use.Flow;
   IF #_w1 THEN #Alarm_SP := #Flow_Line / #SP_M; END_IF;
   #Timers_Alm[0].Start := #_w1 AND (#Alarm_SP < #PID.Converter.Min_Out) AND NOT "Reset_All";
   IF #_w1 AND (#Alarm_SP < #PID.Converter.Min_Out) AND NOT "Reset_All" AND #Timers_Alm[0]."Exit" THEN
       "Alm_Logick" := TRUE;
       #Messages.Low_Duct := TRUE;
       #Messages.Alarm := #Messages.Alarm OR 2#100;
   END_IF;
   #Timers_Stop[0].Start := #Start AND #Messages.Low_Duct AND #Messages_Stop.Low_Duct AND NOT #Messages_Cancel.Low_Duct AND #Timers_Alm[0]."Exit";
   IF NOT #Start OR ((#Alarm_SP > #PID.Converter.Min_Out) AND NOT #PID.CMD.Hand) THEN
       #Messages_Cancel.Low_Duct := FALSE;
   END_IF;
END_REGION

REGION Network 29: Авария - низкий проток
   RUNG wire#powerrail
      Contact( "Reset_All" )
      R_Coil( #Messages_Cancel.Low_Duct )
      R_Coil( #Messages.Low_Duct )
   END_RUNG
   RUNG wire#powerrail
      Contact( #Messages.Low_Duct )
      Contact( #Messages_Stop.Low_Duct )
      I_Contact( #Messages_Cancel.Low_Duct )
      Coil( #Messages_REQ_Stop.Low_Duct )
   END_RUNG
   RUNG wire#powerrail
      P_Contact(operand := #Messages.Low_Duct, bit := #pos[0])
      Add(in1 := #Messages_Counter.Low_Duct, in2 := 1, out => #Messages_Counter.Low_Duct)
   END_RUNG
   RUNG wire#powerrail
      Contact( #Messages_Reset.Low_Duct )
      Move(in := 0, out1 => #Messages_Counter.Low_Duct)
      R_Coil( #Messages_Reset.Low_Duct )
   END_RUNG
   // the same network as SCL:
   IF "Reset_All" THEN
       #Messages_Cancel.Low_Duct := FALSE;
       #Messages.Low_Duct := FALSE;
   END_IF;
   #Messages_REQ_Stop.Low_Duct := #Messages.Low_Duct AND #Messages_Stop.Low_Duct AND NOT #Messages_Cancel.Low_Duct;
   #_w1 := #Messages.Low_Duct AND NOT #pos[0];   // rising edge of #Messages.Low_Duct
   #pos[0] := #Messages.Low_Duct;
   IF #_w1 THEN #Messages_Counter.Low_Duct := #Messages_Counter.Low_Duct + 1; END_IF;
   IF #Messages_Reset.Low_Duct THEN
       #Messages_Counter.Low_Duct := 0;
       #Messages_Reset.Low_Duct := FALSE;
   END_IF;
END_REGION

REGION Network 30: 4. Авария - нет ротаметра
   #Timers_Alm[2].Start := #Start AND #Mode AND #Use.RT AND #KC_CMD AND NOT #RT AND NOT "Reset_All";
   IF #Start AND #Mode AND #Use.RT AND #KC_CMD AND NOT #RT AND NOT "Reset_All" AND #Timers_Alm[2]."Exit" THEN
       "Alm_Logick" := TRUE;
       #Messages.RT_ON := TRUE;
       #Messages.Alarm := #Messages.Alarm OR 2#1000;
   END_IF;
   #Timers_Stop[2].Start := #Start AND #Messages.RT_ON AND #Messages_Stop.RT_ON AND NOT #Messages_Cancel.RT_ON AND #Timers_Alm[2]."Exit";
   IF NOT #Start OR #RT THEN #Messages_Cancel.RT_ON := FALSE; END_IF;
END_REGION

REGION Network 31: Авария - нет ротаметра
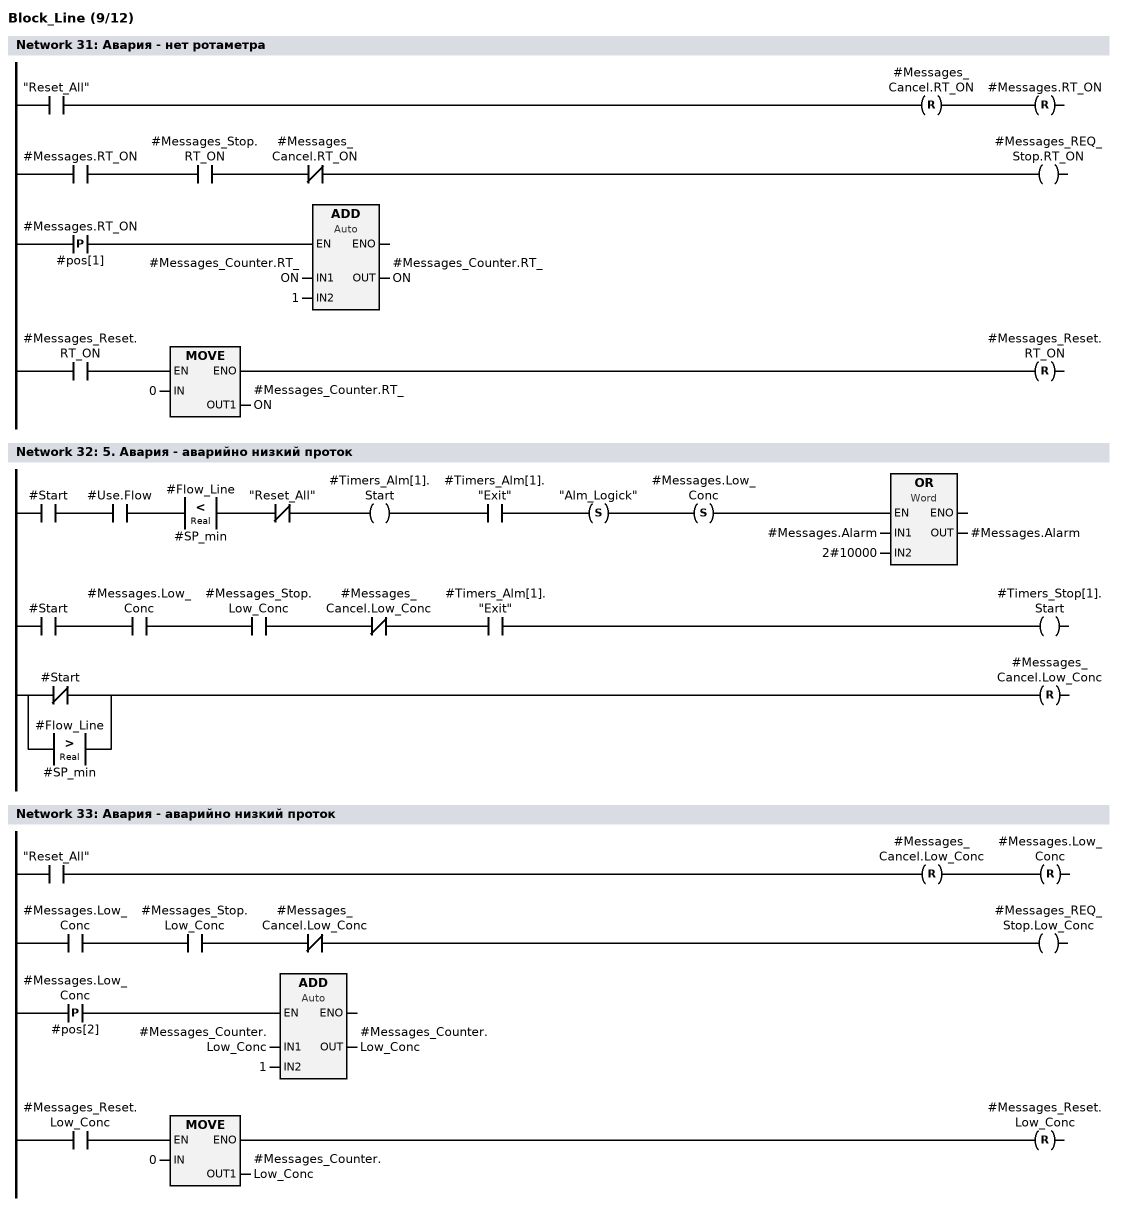
   RUNG wire#powerrail
      Contact( "Reset_All" )
      R_Coil( #Messages_Cancel.RT_ON )
      R_Coil( #Messages.RT_ON )
   END_RUNG
   RUNG wire#powerrail
      Contact( #Messages.RT_ON )
      Contact( #Messages_Stop.RT_ON )
      I_Contact( #Messages_Cancel.RT_ON )
      Coil( #Messages_REQ_Stop.RT_ON )
   END_RUNG
   RUNG wire#powerrail
      P_Contact(operand := #Messages.RT_ON, bit := #pos[1])
      Add(in1 := #Messages_Counter.RT_ON, in2 := 1, out => #Messages_Counter.RT_ON)
   END_RUNG
   RUNG wire#powerrail
      Contact( #Messages_Reset.RT_ON )
      Move(in := 0, out1 => #Messages_Counter.RT_ON)
      R_Coil( #Messages_Reset.RT_ON )
   END_RUNG
   // the same network as SCL:
   IF "Reset_All" THEN
       #Messages_Cancel.RT_ON := FALSE;
       #Messages.RT_ON := FALSE;
   END_IF;
   #Messages_REQ_Stop.RT_ON := #Messages.RT_ON AND #Messages_Stop.RT_ON AND NOT #Messages_Cancel.RT_ON;
   #_w1 := #Messages.RT_ON AND NOT #pos[1];   // rising edge of #Messages.RT_ON
   #pos[1] := #Messages.RT_ON;
   IF #_w1 THEN #Messages_Counter.RT_ON := #Messages_Counter.RT_ON + 1; END_IF;
   IF #Messages_Reset.RT_ON THEN
       #Messages_Counter.RT_ON := 0;
       #Messages_Reset.RT_ON := FALSE;
   END_IF;
END_REGION

REGION Network 32: 5. Авария - аварийно низкий проток
   #Timers_Alm[1].Start := #Start AND #Use.Flow AND (#Flow_Line < #SP_min) AND NOT "Reset_All";
   IF #Start AND #Use.Flow AND (#Flow_Line < #SP_min) AND NOT "Reset_All" AND #Timers_Alm[1]."Exit" THEN
       "Alm_Logick" := TRUE;
       #Messages.Low_Conc := TRUE;
       #Messages.Alarm := #Messages.Alarm OR 2#10000;
   END_IF;
   #Timers_Stop[1].Start := #Start AND #Messages.Low_Conc AND #Messages_Stop.Low_Conc AND NOT #Messages_Cancel.Low_Conc AND #Timers_Alm[1]."Exit";
   IF NOT #Start OR (#Flow_Line > #SP_min) THEN #Messages_Cancel.Low_Conc := FALSE; END_IF;
END_REGION

REGION Network 33: Авария - аварийно низкий проток
   RUNG wire#powerrail
      Contact( "Reset_All" )
      R_Coil( #Messages_Cancel.Low_Conc )
      R_Coil( #Messages.Low_Conc )
   END_RUNG
   RUNG wire#powerrail
      Contact( #Messages.Low_Conc )
      Contact( #Messages_Stop.Low_Conc )
      I_Contact( #Messages_Cancel.Low_Conc )
      Coil( #Messages_REQ_Stop.Low_Conc )
   END_RUNG
   RUNG wire#powerrail
      P_Contact(operand := #Messages.Low_Conc, bit := #pos[2])
      Add(in1 := #Messages_Counter.Low_Conc, in2 := 1, out => #Messages_Counter.Low_Conc)
   END_RUNG
   RUNG wire#powerrail
      Contact( #Messages_Reset.Low_Conc )
      Move(in := 0, out1 => #Messages_Counter.Low_Conc)
      R_Coil( #Messages_Reset.Low_Conc )
   END_RUNG
   // the same network as SCL:
   IF "Reset_All" THEN
       #Messages_Cancel.Low_Conc := FALSE;
       #Messages.Low_Conc := FALSE;
   END_IF;
   #Messages_REQ_Stop.Low_Conc := #Messages.Low_Conc AND #Messages_Stop.Low_Conc AND NOT #Messages_Cancel.Low_Conc;
   #_w1 := #Messages.Low_Conc AND NOT #pos[2];   // rising edge of #Messages.Low_Conc
   #pos[2] := #Messages.Low_Conc;
   IF #_w1 THEN #Messages_Counter.Low_Conc := #Messages_Counter.Low_Conc + 1; END_IF;
   IF #Messages_Reset.Low_Conc THEN
       #Messages_Counter.Low_Conc := 0;
       #Messages_Reset.Low_Conc := FALSE;
   END_IF;
END_REGION

REGION Network 34: 6. Авария - застрял ротаметр
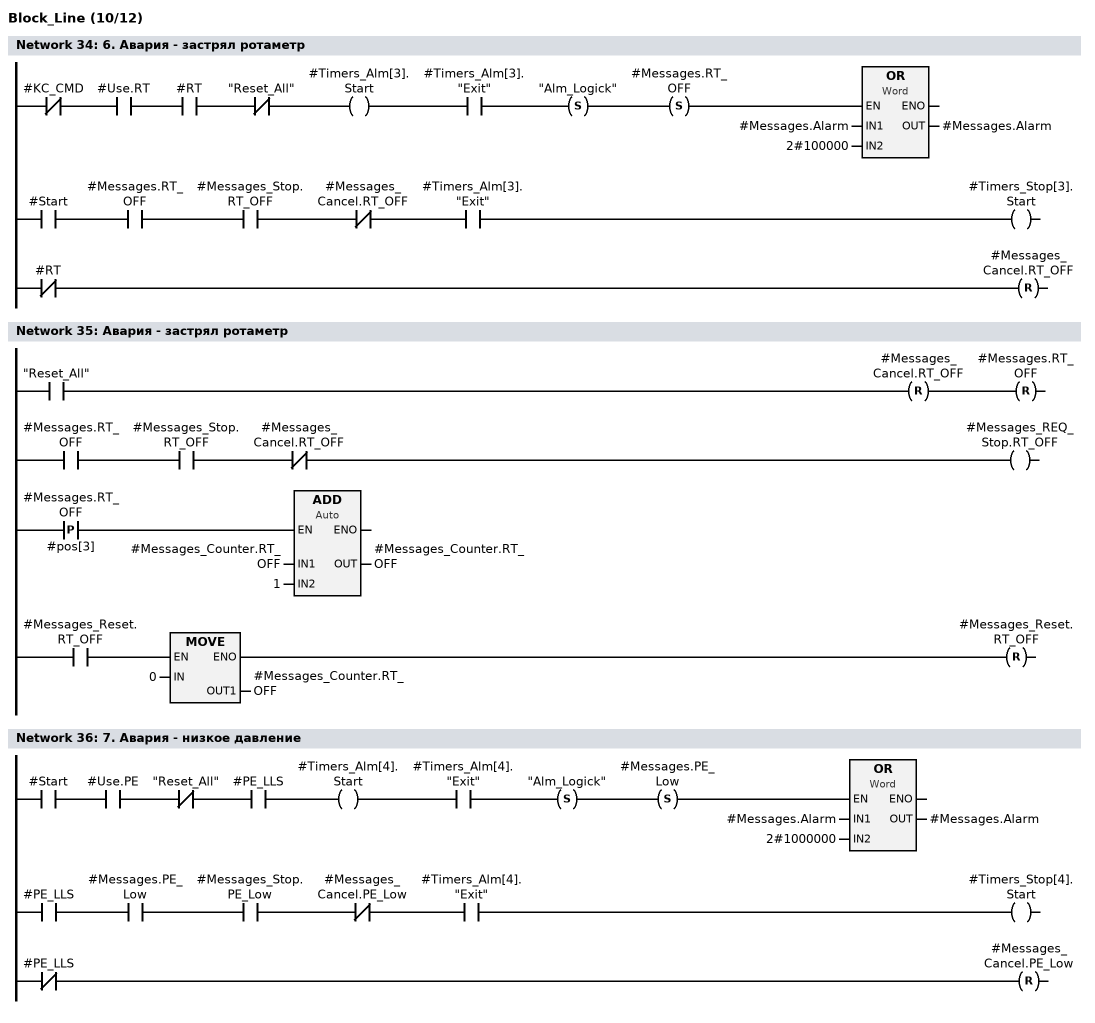
   #Timers_Alm[3].Start := NOT #KC_CMD AND #Use.RT AND #RT AND NOT "Reset_All";
   IF NOT #KC_CMD AND #Use.RT AND #RT AND NOT "Reset_All" AND #Timers_Alm[3]."Exit" THEN
       "Alm_Logick" := TRUE;
       #Messages.RT_OFF := TRUE;
       #Messages.Alarm := #Messages.Alarm OR 2#100000;
   END_IF;
   #Timers_Stop[3].Start := #Start AND #Messages.RT_OFF AND #Messages_Stop.RT_OFF AND NOT #Messages_Cancel.RT_OFF AND #Timers_Alm[3]."Exit";
   IF NOT #RT THEN #Messages_Cancel.RT_OFF := FALSE; END_IF;
END_REGION

REGION Network 35: Авария - застрял ротаметр
   RUNG wire#powerrail
      Contact( "Reset_All" )
      R_Coil( #Messages_Cancel.RT_OFF )
      R_Coil( #Messages.RT_OFF )
   END_RUNG
   RUNG wire#powerrail
      Contact( #Messages.RT_OFF )
      Contact( #Messages_Stop.RT_OFF )
      I_Contact( #Messages_Cancel.RT_OFF )
      Coil( #Messages_REQ_Stop.RT_OFF )
   END_RUNG
   RUNG wire#powerrail
      P_Contact(operand := #Messages.RT_OFF, bit := #pos[3])
      Add(in1 := #Messages_Counter.RT_OFF, in2 := 1, out => #Messages_Counter.RT_OFF)
   END_RUNG
   RUNG wire#powerrail
      Contact( #Messages_Reset.RT_OFF )
      Move(in := 0, out1 => #Messages_Counter.RT_OFF)
      R_Coil( #Messages_Reset.RT_OFF )
   END_RUNG
   // the same network as SCL:
   IF "Reset_All" THEN
       #Messages_Cancel.RT_OFF := FALSE;
       #Messages.RT_OFF := FALSE;
   END_IF;
   #Messages_REQ_Stop.RT_OFF := #Messages.RT_OFF AND #Messages_Stop.RT_OFF AND NOT #Messages_Cancel.RT_OFF;
   #_w1 := #Messages.RT_OFF AND NOT #pos[3];   // rising edge of #Messages.RT_OFF
   #pos[3] := #Messages.RT_OFF;
   IF #_w1 THEN #Messages_Counter.RT_OFF := #Messages_Counter.RT_OFF + 1; END_IF;
   IF #Messages_Reset.RT_OFF THEN
       #Messages_Counter.RT_OFF := 0;
       #Messages_Reset.RT_OFF := FALSE;
   END_IF;
END_REGION

REGION Network 36: 7. Авария - низкое давление
   #Timers_Alm[4].Start := #Start AND #Use.PE AND NOT "Reset_All" AND #PE_LLS;
   IF #Start AND #Use.PE AND NOT "Reset_All" AND #PE_LLS AND #Timers_Alm[4]."Exit" THEN
       "Alm_Logick" := TRUE;
       #Messages.PE_Low := TRUE;
       #Messages.Alarm := #Messages.Alarm OR 2#1000000;
   END_IF;
   #Timers_Stop[4].Start := #PE_LLS AND #Messages.PE_Low AND #Messages_Stop.PE_Low AND NOT #Messages_Cancel.PE_Low AND #Timers_Alm[4]."Exit";
   IF NOT #PE_LLS THEN #Messages_Cancel.PE_Low := FALSE; END_IF;
END_REGION

REGION Network 37: Авария - низкое давление
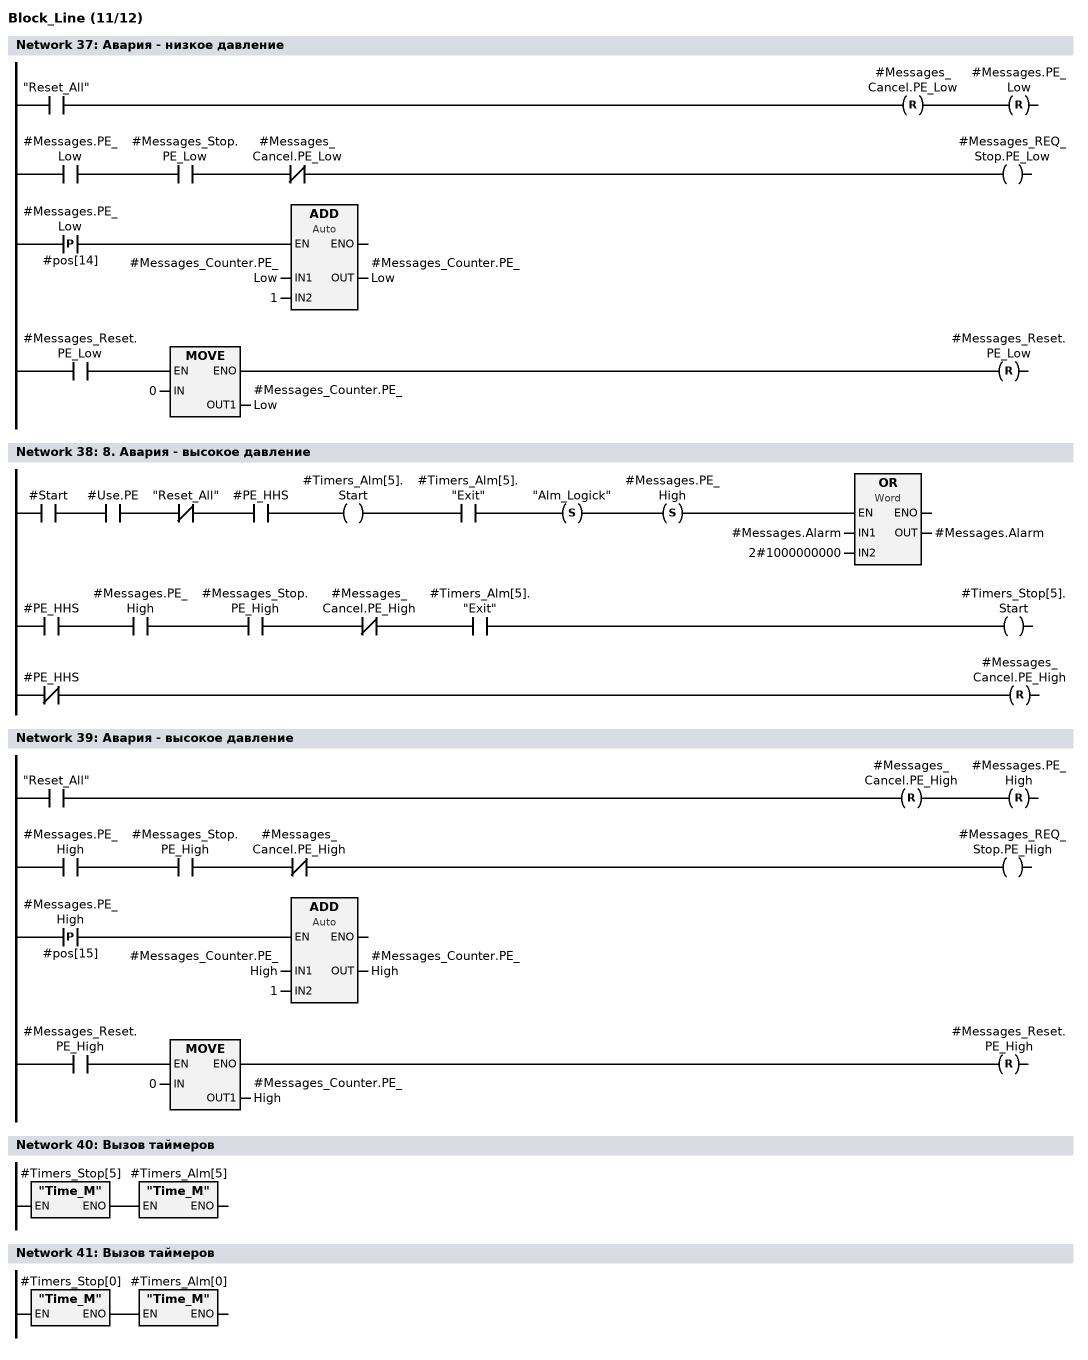
   RUNG wire#powerrail
      Contact( "Reset_All" )
      R_Coil( #Messages_Cancel.PE_Low )
      R_Coil( #Messages.PE_Low )
   END_RUNG
   RUNG wire#powerrail
      Contact( #Messages.PE_Low )
      Contact( #Messages_Stop.PE_Low )
      I_Contact( #Messages_Cancel.PE_Low )
      Coil( #Messages_REQ_Stop.PE_Low )
   END_RUNG
   RUNG wire#powerrail
      P_Contact(operand := #Messages.PE_Low, bit := #pos[14])
      Add(in1 := #Messages_Counter.PE_Low, in2 := 1, out => #Messages_Counter.PE_Low)
   END_RUNG
   RUNG wire#powerrail
      Contact( #Messages_Reset.PE_Low )
      Move(in := 0, out1 => #Messages_Counter.PE_Low)
      R_Coil( #Messages_Reset.PE_Low )
   END_RUNG
   // the same network as SCL:
   IF "Reset_All" THEN
       #Messages_Cancel.PE_Low := FALSE;
       #Messages.PE_Low := FALSE;
   END_IF;
   #Messages_REQ_Stop.PE_Low := #Messages.PE_Low AND #Messages_Stop.PE_Low AND NOT #Messages_Cancel.PE_Low;
   #_w1 := #Messages.PE_Low AND NOT #pos[14];   // rising edge of #Messages.PE_Low
   #pos[14] := #Messages.PE_Low;
   IF #_w1 THEN #Messages_Counter.PE_Low := #Messages_Counter.PE_Low + 1; END_IF;
   IF #Messages_Reset.PE_Low THEN
       #Messages_Counter.PE_Low := 0;
       #Messages_Reset.PE_Low := FALSE;
   END_IF;
END_REGION

REGION Network 38: 8. Авария - высокое давление
   #Timers_Alm[5].Start := #Start AND #Use.PE AND NOT "Reset_All" AND #PE_HHS;
   IF #Start AND #Use.PE AND NOT "Reset_All" AND #PE_HHS AND #Timers_Alm[5]."Exit" THEN
       "Alm_Logick" := TRUE;
       #Messages.PE_High := TRUE;
       #Messages.Alarm := #Messages.Alarm OR 2#1000000000;
   END_IF;
   #Timers_Stop[5].Start := #PE_HHS AND #Messages.PE_High AND #Messages_Stop.PE_High AND NOT #Messages_Cancel.PE_High AND #Timers_Alm[5]."Exit";
   IF NOT #PE_HHS THEN #Messages_Cancel.PE_High := FALSE; END_IF;
END_REGION

REGION Network 39: Авария - высокое давление
   RUNG wire#powerrail
      Contact( "Reset_All" )
      R_Coil( #Messages_Cancel.PE_High )
      R_Coil( #Messages.PE_High )
   END_RUNG
   RUNG wire#powerrail
      Contact( #Messages.PE_High )
      Contact( #Messages_Stop.PE_High )
      I_Contact( #Messages_Cancel.PE_High )
      Coil( #Messages_REQ_Stop.PE_High )
   END_RUNG
   RUNG wire#powerrail
      P_Contact(operand := #Messages.PE_High, bit := #pos[15])
      Add(in1 := #Messages_Counter.PE_High, in2 := 1, out => #Messages_Counter.PE_High)
   END_RUNG
   RUNG wire#powerrail
      Contact( #Messages_Reset.PE_High )
      Move(in := 0, out1 => #Messages_Counter.PE_High)
      R_Coil( #Messages_Reset.PE_High )
   END_RUNG
   // the same network as SCL:
   IF "Reset_All" THEN
       #Messages_Cancel.PE_High := FALSE;
       #Messages.PE_High := FALSE;
   END_IF;
   #Messages_REQ_Stop.PE_High := #Messages.PE_High AND #Messages_Stop.PE_High AND NOT #Messages_Cancel.PE_High;
   #_w1 := #Messages.PE_High AND NOT #pos[15];   // rising edge of #Messages.PE_High
   #pos[15] := #Messages.PE_High;
   IF #_w1 THEN #Messages_Counter.PE_High := #Messages_Counter.PE_High + 1; END_IF;
   IF #Messages_Reset.PE_High THEN
       #Messages_Counter.PE_High := 0;
       #Messages_Reset.PE_High := FALSE;
   END_IF;
END_REGION

REGION Network 40: Вызов таймеров
   RUNG wire#powerrail
      #Timers_Stop[5]()
      #Timers_Alm[5]()
   END_RUNG
   // the same network as SCL:
   #Timers_Stop[5](ENO => #_w1);   // "Time_M"
   IF #_w1 THEN
       #Timers_Alm[5]();   // "Time_M"
   END_IF;
END_REGION

REGION Network 41: Вызов таймеров
   RUNG wire#powerrail
      #Timers_Stop[0]()
      #Timers_Alm[0]()
   END_RUNG
   // the same network as SCL:
   #Timers_Stop[0](ENO => #_w1);   // "Time_M"
   IF #_w1 THEN
       #Timers_Alm[0]();   // "Time_M"
   END_IF;
END_REGION

REGION Network 42: Вызов таймеров
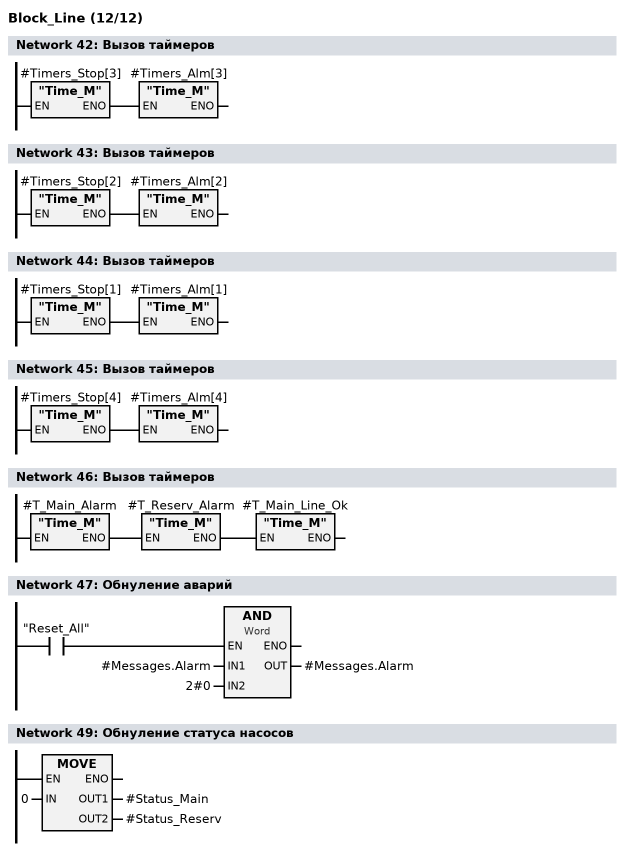
   RUNG wire#powerrail
      #Timers_Stop[3]()
      #Timers_Alm[3]()
   END_RUNG
   // the same network as SCL:
   #Timers_Stop[3](ENO => #_w1);   // "Time_M"
   IF #_w1 THEN
       #Timers_Alm[3]();   // "Time_M"
   END_IF;
END_REGION

REGION Network 43: Вызов таймеров
   RUNG wire#powerrail
      #Timers_Stop[2]()
      #Timers_Alm[2]()
   END_RUNG
   // the same network as SCL:
   #Timers_Stop[2](ENO => #_w1);   // "Time_M"
   IF #_w1 THEN
       #Timers_Alm[2]();   // "Time_M"
   END_IF;
END_REGION

REGION Network 44: Вызов таймеров
   RUNG wire#powerrail
      #Timers_Stop[1]()
      #Timers_Alm[1]()
   END_RUNG
   // the same network as SCL:
   #Timers_Stop[1](ENO => #_w1);   // "Time_M"
   IF #_w1 THEN
       #Timers_Alm[1]();   // "Time_M"
   END_IF;
END_REGION

REGION Network 45: Вызов таймеров
   RUNG wire#powerrail
      #Timers_Stop[4]()
      #Timers_Alm[4]()
   END_RUNG
   // the same network as SCL:
   #Timers_Stop[4](ENO => #_w1);   // "Time_M"
   IF #_w1 THEN
       #Timers_Alm[4]();   // "Time_M"
   END_IF;
END_REGION

REGION Network 46: Вызов таймеров
   RUNG wire#powerrail
      #T_Main_Alarm()
      #T_Reserv_Alarm()
      #T_Main_Line_Ok()
   END_RUNG
   // the same network as SCL:
   #T_Main_Alarm(ENO => #_w1);   // "Time_M"
   #T_Reserv_Alarm(EN := #_w1, ENO => #_w2);   // "Time_M"
   IF #_w2 THEN
       #T_Main_Line_Ok();   // "Time_M"
   END_IF;
END_REGION

REGION Network 47: Обнуление аварий
   RUNG wire#powerrail
      Contact( "Reset_All" )
      { S7_Templates := "SrcType := Word" } And(in1 := #Messages.Alarm, in2 := 2#0, out => #Messages.Alarm)
   END_RUNG
   // the same network as SCL:
   IF "Reset_All" THEN #Messages.Alarm := #Messages.Alarm AND 2#0; END_IF;
END_REGION

REGION Network 48: Обнуление Report
END_REGION

REGION Network 49: Обнуление статуса насосов
   RUNG wire#powerrail
      Move(in := 0, out1 => #Status_Main, out2 => #Status_Reserv)
   END_RUNG
   // the same network as SCL:
   #Status_Main := 0;
   #Status_Reserv := 0;
END_REGION
END_FUNCTION_BLOCK
